LIN {X 0,Y 234.261,Z 267.411,A -85,B 0,C 180,E1 -19867.278,E2 -19867.278} C_VEL
LIN {X 0,Y 232.34,Z 276.851,A -85,B 0,C 180,E1 -19869.181,E2 -19869.181} C_VEL
LIN {X 0,Y 230.576,Z 285.695,A -85,B 0,C 180,E1 -19871.384,E2 -19871.384} C_VEL
LIN {X 0,Y 228.899,Z 293.962,A -85,B 0,C 180,E1 -19873.959,E2 -19873.959} C_VEL
LIN {X 0,Y 227.464,Z 300.726,A -85,B 0,C 180,E1 -19876.601,E2 -19876.601} C_VEL
LIN {X 0,Y 226.631,Z 306.146,A -85,B 0,C 180,E1 -19879.277,E2 -19879.277} C_VEL
LIN {X 0,Y 226.113,Z 310.355,A -85,B 0,C 180,E1 -19881.96,E2 -19881.96} C_VEL
LIN {X 0,Y 225.925,Z 313.474,A -85,B 0,C 180,E1 -19884.645,E2 -19884.645} C_VEL
LIN {X 0,Y 225.892,Z 315.003,A -85,B 0,C 180,E1 -19886.433,E2 -19886.433} C_VEL
LIN {X 0,Y 225.898,Z 316.083,A -85,B 0,C 180,E1 -19888.217,E2 -19888.217} C_VEL
LIN {X 0,Y 225.948,Z 316.728,A -85,B 0,C 180,E1 -19890,E2 -19890} C_VEL
LIN {X 0,Y 225.881,Z 316.964,A -85,B 0,C 180,E1 -19891.783,E2 -19891.783} C_VEL
LIN {X 0,Y 225.778,Z 316.356,A -85,B 0,C 180,E1 -19895.057,E2 -19895.057} C_VEL
LIN {X 0,Y 225.93,Z 315.246,A -85,B 0,C 180,E1 -19897.148,E2 -19897.148} C_VEL
LIN {X 0,Y 226.587,Z 312.1,A -85,B 0,C 180,E1 -19900.726,E2 -19900.726} C_VEL
LIN {X 0,Y 227.542,Z 308.619,A -85,B 0,C 180,E1 -19903.395,E2 -19903.395} C_VEL
LIN {X 0,Y 229.085,Z 304.112,A -85,B 0,C 180,E1 -19906.028,E2 -19906.028} C_VEL
LIN {X 0,Y 231.41,Z 297.415,A -85,B 0,C 180,E1 -19909.056,E2 -19909.056} C_VEL
LIN {X 0,Y 233.842,Z 290.185,A -85,B 0,C 180,E1 -19911.603,E2 -19911.603} C_VEL
LIN {X 0,Y 236.778,Z 281.363,A -85,B 0,C 180,E1 -19914.087,E2 -19914.087} C_VEL
LIN {X 0,Y 239.631,Z 272.445,A -85,B 0,C 180,E1 -19916.1,E2 -19916.1} C_VEL
LIN {X 0,Y 240.939,Z 262.483,A -85,B 0,C 180,E1 -19918.163,E2 -19918.163} C_VEL
LIN {X 0,Y 241.294,Z 252.576,A -85,B 0,C 180,E1 -19920.006,E2 -19920.006} C_VEL
LIN {X 0,Y 240.625,Z 241.498,A -85,B 0,C 180,E1 -19921.938,E2 -19921.938} C_VEL
LIN {X 0,Y 239.232,Z 232.018,A -85,B 0,C 180,E1 -19923.532,E2 -19923.532} C_VEL
LIN {X 0,Y 235.782,Z 218.471,A -85,B 0,C 180,E1 -19925.831,E2 -19925.831} C_VEL
LIN {X 0,Y 234.537,Z 214.79,A -85,B 0,C 180,E1 -19926.496,E2 -19926.496} C_VEL
LIN {X 0,Y 233.156,Z 210.978,A -85,B 0,C 180,E1 -19927.17,E2 -19927.17} C_VEL
LIN {X 0,Y 231.728,Z 207.641,A -85,B 0,C 180,E1 -19927.812,E2 -19927.812} C_VEL
LIN {X 0,Y 231.483,Z 206.301,A -85,B 0,C 180,E1 -19928.038,E2 -19928.038} C_VEL
LIN {X 0,Y 231.379,Z 203.886,A -85,B 0,C 180,E1 -19930.591,E2 -19930.591} C_VEL
LIN {X 0,Y 230.811,Z 200.597,A -85,B 0,C 180,E1 -19934.454,E2 -19934.454} C_VEL
LIN {X 0,Y 230.336,Z 198.024,A -85,B 0,C 180,E1 -19937.834,E2 -19937.834} C_VEL
LIN {X 0,Y 230.103,Z 196.43,A -85,B 0,C 180,E1 -19940.103,E2 -19940.103} C_VEL
LIN {X 0,Y 229.632,Z 193.775,A -85,B 0,C 180,E1 -19944.443,E2 -19944.443} C_VEL
LIN {X 0,Y 229.255,Z 191.689,A -85,B 0,C 180,E1 -19948.59,E2 -19948.59} C_VEL
LIN {X 0,Y 229.015,Z 189.98,A -85,B 0,C 180,E1 -19952.868,E2 -19952.868} C_VEL
LIN {X 0,Y 228.806,Z 188.731,A -85,B 0,C 180,E1 -19957.145,E2 -19957.145} C_VEL
LIN {X 0,Y 228.703,Z 187.823,A -85,B 0,C 180,E1 -19962.294,E2 -19962.294} C_VEL
LIN {X 0,Y 228.699,Z 187.554,A -85,B 0,C 180,E1 -19965.767,E2 -19965.767} C_VEL
LIN {X 0,Y 228.837,Z 187.534,A -85,B 0,C 180,E1 -19969.38,E2 -19969.38} C_VEL
LIN {X 0,Y 228.961,Z 187.798,A -85,B 0,C 180,E1 -19972.946,E2 -19972.946} C_VEL
LIN {X 0,Y 229.333,Z 188.636,A -85,B 0,C 180,E1 -19978.243,E2 -19978.243} C_VEL
LIN {X 0,Y 229.495,Z 189.026,A -85,B 0,C 180,E1 -19979.999,E2 -19979.999} C_VEL
LIN {X 0,Y 229.331,Z 190.067,A -85,B 0,C 180,E1 -19983.513,E2 -19983.513} C_VEL
LIN {X 0,Y 229.34,Z 191.116,A -85,B 0,C 180,E1 -19986.598,E2 -19986.598} C_VEL
LIN {X 0,Y 230.655,Z 194.258,A -85,B 0,C 180,E1 -19987.275,E2 -19987.275} C_VEL
LIN {X 0,Y 232.372,Z 196.596,A -85,B 0,C 180,E1 -19987.985,E2 -19987.985} C_VEL
LIN {X 0,Y 234.252,Z 199.958,A -85,B 0,C 180,E1 -19988.842,E2 -19988.842} C_VEL
LIN {X 0,Y 238.567,Z 209.506,A -85,B 0,C 180,E1 -19991.039,E2 -19991.039} C_VEL
LIN {X 0,Y 241.815,Z 218.493,A -85,B 0,C 180,E1 -19993.016,E2 -19993.016} C_VEL
LIN {X 0,Y 244.147,Z 227.757,A -85,B 0,C 180,E1 -19995.014,E2 -19995.014} C_VEL
LIN {X 0,Y 245.461,Z 237.244,A -85,B 0,C 180,E1 -19997.065,E2 -19997.065} C_VEL
LIN {X 0,Y 245.251,Z 239.564,A -85,B 0,C 180,E1 -19997.51,E2 -19997.51} C_VEL
LIN {X 0,Y 242.506,Z 249.033,A -85,B 0,C 180,E1 -19999.247,E2 -19999.247} C_VEL
LIN {X 0,Y 239.388,Z 258.851,A -85,B 0,C 180,E1 -20001.545,E2 -20001.545} C_VEL
LIN {X 0,Y 236.513,Z 266.907,A -85,B 0,C 180,E1 -20003.899,E2 -20003.899} C_VEL
LIN {X 0,Y 234.073,Z 273.398,A -85,B 0,C 180,E1 -20006.289,E2 -20006.289} C_VEL
LIN {X 0,Y 231.665,Z 279.237,A -85,B 0,C 180,E1 -20009.037,E2 -20009.037} C_VEL
LIN {X 0,Y 230.067,Z 282.963,A -85,B 0,C 180,E1 -20011.285,E2 -20011.285} C_VEL
LIN {X 0,Y 228.599,Z 286.233,A -85,B 0,C 180,E1 -20013.892,E2 -20013.892} C_VEL
LIN {X 0,Y 227.452,Z 288.559,A -85,B 0,C 180,E1 -20016.546,E2 -20016.546} C_VEL
LIN {X 0,Y 226.601,Z 289.931,A -85,B 0,C 180,E1 -20019.16,E2 -20019.16} C_VEL
LIN {X 0,Y 226.076,Z 290.434,A -85,B 0,C 180,E1 -20021.747,E2 -20021.747} C_VEL
LIN {X 0,Y 225.813,Z 290.119,A -85,B 0,C 180,E1 -20024.288,E2 -20024.288} C_VEL
LIN {X 0,Y 225.802,Z 289.027,A -85,B 0,C 180,E1 -20026.784,E2 -20026.784} C_VEL
LIN {X 0,Y 226.011,Z 287.146,A -85,B 0,C 180,E1 -20029.23,E2 -20029.23} C_VEL
LIN {X 0,Y 226.502,Z 284.502,A -85,B 0,C 180,E1 -20031.642,E2 -20031.642} C_VEL
LIN {X 0,Y 227.12,Z 281.132,A -85,B 0,C 180,E1 -20033.989,E2 -20033.989} C_VEL
LIN {X 0,Y 228.162,Z 275.652,A -85,B 0,C 180,E1 -20036.911,E2 -20036.911} C_VEL
LIN {X 0,Y 229.37,Z 269.303,A -85,B 0,C 180,E1 -20039.562,E2 -20039.562} C_VEL
LIN {X 0,Y 230.885,Z 262.103,A -85,B 0,C 180,E1 -20041.973,E2 -20041.973} C_VEL
LIN {X 0,Y 232.717,Z 252.954,A -85,B 0,C 180,E1 -20044.431,E2 -20044.431} C_VEL
LIN {X 0,Y 234.58,Z 242.855,A -85,B 0,C 180,E1 -20046.611,E2 -20046.611} C_VEL
LIN {X 0,Y 236.408,Z 232.431,A -85,B 0,C 180,E1 -20048.414,E2 -20048.414} C_VEL
LIN {X 0,Y 237.204,Z 227.255,A -85,B 0,C 180,E1 -20049.173,E2 -20049.173} C_VEL
LIN {X 0,Y 235.754,Z 217.735,A -85,B 0,C 180,E1 -20050.631,E2 -20050.631} C_VEL
LIN {X 0,Y 233.026,Z 205.757,A -85,B 0,C 180,E1 -20052.232,E2 -20052.232} C_VEL
LIN {X 0,Y 229.467,Z 193.019,A -85,B 0,C 180,E1 -20053.655,E2 -20053.655} C_VEL
LIN {X 0,Y 227.315,Z 185.716,A -85,B 0,C 180,E1 -20054.361,E2 -20054.361} C_VEL
LIN {X 0,Y 227.348,Z 184.804,A -85,B 0,C 180,E1 -20055.682,E2 -20055.682} C_VEL
LIN {X 0,Y 227.548,Z 184.141,A -85,B 0,C 180,E1 -20057.514,E2 -20057.514} C_VEL
LIN {X 0,Y 228.127,Z 184.067,A -85,B 0,C 180,E1 -20061.139,E2 -20061.139} C_VEL
LIN {X 0,Y 228.274,Z 184.051,A -85,B 0,C 180,E1 -20062.926,E2 -20062.926} C_VEL
LIN {X 0,Y 228.552,Z 184.018,A -85,B 0,C 180,E1 -20068.238,E2 -20068.238} C_VEL
LIN {X 0,Y 228.552,Z 184.014,A -85,B 0,C 180,E1 -20071.762,E2 -20071.762} C_VEL
LIN {X 0,Y 228.355,Z 184.04,A -85,B 0,C 180,E1 -20077.071,E2 -20077.071} C_VEL
LIN {X 0,Y 228.169,Z 184.059,A -85,B 0,C 180,E1 -20080.65,E2 -20080.65} C_VEL
LIN {X 0,Y 228.055,Z 184.078,A -85,B 0,C 180,E1 -20086.102,E2 -20086.102} C_VEL
LIN {X 0,Y 227.951,Z 184.094,A -85,B 0,C 180,E1 -20089.824,E2 -20089.824} C_VEL
LIN {X 0,Y 227.921,Z 184.096,A -85,B 0,C 180,E1 -20093.632,E2 -20093.632} C_VEL
LIN {X 0,Y 227.876,Z 184.097,A -85,B 0,C 180,E1 -20097.556,E2 -20097.556} C_VEL
LIN {X 0,Y 227.863,Z 184.102,A -85,B 0,C 180,E1 -20101.623,E2 -20101.623} C_VEL
LIN {X 0,Y 227.877,Z 184.091,A -85,B 0,C 180,E1 -20105.872,E2 -20105.872} C_VEL
LIN {X 0,Y 227.824,Z 184.104,A -85,B 0,C 180,E1 -20110.377,E2 -20110.377} C_VEL
LIN {X 0,Y 227.833,Z 184.102,A -85,B 0,C 180,E1 -20115.193,E2 -20115.193} C_VEL
LIN {X 0,Y 227.824,Z 184.099,A -85,B 0,C 180,E1 -20119.624,E2 -20119.624} C_VEL
LIN {X 0,Y 227.878,Z 184.098,A -85,B 0,C 180,E1 -20124.129,E2 -20124.129} C_VEL
LIN {X 0,Y 227.865,Z 184.098,A -85,B 0,C 180,E1 -20128.378,E2 -20128.378} C_VEL
LIN {X 0,Y 227.878,Z 184.09,A -85,B 0,C 180,E1 -20132.445,E2 -20132.445} C_VEL
LIN {X 0,Y 227.924,Z 184.093,A -85,B 0,C 180,E1 -20136.37,E2 -20136.37} C_VEL
LIN {X 0,Y 227.954,Z 184.089,A -85,B 0,C 180,E1 -20140.177,E2 -20140.177} C_VEL
LIN {X 0,Y 228.058,Z 184.067,A -85,B 0,C 180,E1 -20143.899,E2 -20143.899} C_VEL
LIN {X 0,Y 228.073,Z 184.069,A -85,B 0,C 180,E1 -20147.544,E2 -20147.544} C_VEL
LIN {X 0,Y 228.268,Z 184.049,A -85,B 0,C 180,E1 -20151.145,E2 -20151.145} C_VEL
LIN {X 0,Y 228.325,Z 184.041,A -85,B 0,C 180,E1 -20152.929,E2 -20152.929} C_VEL
LIN {X 0,Y 228.556,Z 184.007,A -85,B 0,C 180,E1 -20158.239,E2 -20158.239} C_VEL
LIN {X 0,Y 228.554,Z 184.014,A -85,B 0,C 180,E1 -20161.763,E2 -20161.763} C_VEL
LIN {X 0,Y 228.312,Z 184.04,A -85,B 0,C 180,E1 -20167.074,E2 -20167.074} C_VEL
LIN {X 0,Y 228.147,Z 184.062,A -85,B 0,C 180,E1 -20170.652,E2 -20170.652} C_VEL
LIN {X 0,Y 228.066,Z 184.075,A -85,B 0,C 180,E1 -20174.273,E2 -20174.273} C_VEL
LIN {X 0,Y 228.009,Z 184.079,A -85,B 0,C 180,E1 -20177.954,E2 -20177.954} C_VEL
LIN {X 0,Y 227.962,Z 184.087,A -85,B 0,C 180,E1 -20182.349,E2 -20182.349} C_VEL
LIN {X 0,Y 227.944,Z 184.091,A -85,B 0,C 180,E1 -20186.603,E2 -20186.603} C_VEL
LIN {X 0,Y 227.899,Z 184.096,A -85,B 0,C 180,E1 -20190.292,E2 -20190.292} C_VEL
LIN {X 0,Y 227.924,Z 184.095,A -85,B 0,C 180,E1 -20195.593,E2 -20195.593} C_VEL
LIN {X 0,Y 228.305,Z 186.122,A -85,B 0,C 180,E1 -20198.002,E2 -20198.002} C_VEL
LIN {X 0,Y 229.05,Z 190.541,A -85,B 0,C 180,E1 -20202.575,E2 -20202.575} C_VEL
LIN {X 0,Y 229.95,Z 195.263,A -85,B 0,C 180,E1 -20207.183,E2 -20207.183} C_VEL
LIN {X 0,Y 230.531,Z 198.513,A -85,B 0,C 180,E1 -20210.193,E2 -20210.193} C_VEL
LIN {X 0,Y 230.681,Z 201.082,A -85,B 0,C 180,E1 -20212.459,E2 -20212.459} C_VEL
LIN {X 0,Y 230.036,Z 204.782,A -85,B 0,C 180,E1 -20215.579,E2 -20215.579} C_VEL
LIN {X 0,Y 228.719,Z 210.452,A -85,B 0,C 180,E1 -20220.196,E2 -20220.196} C_VEL
LIN {X 0,Y 235.294,Z 214.381,A -85,B 0,C 180,E1 -20221.089,E2 -20221.089} C_VEL
LIN {X 0,Y 236.925,Z 216.569,A -85,B 0,C 180,E1 -20221.397,E2 -20221.397} C_VEL
LIN {X 0,Y 237.155,Z 218.575,A -85,B 0,C 180,E1 -20221.524,E2 -20221.524} C_VEL
LIN {X 0,Y 236.001,Z 220.936,A -85,B 0,C 180,E1 -20221.537,E2 -20221.537} C_VEL
LIN {X 0,Y 229.339,Z 226.777,A -85,B 0,C 180,E1 -20221.396,E2 -20221.396} C_VEL
LIN {X 0,Y 228.283,Z 229.366,A -85,B 0,C 180,E1 -20221.512,E2 -20221.512} C_VEL
LIN {X 0,Y 227.469,Z 232.667,A -85,B 0,C 180,E1 -20221.765,E2 -20221.765} C_VEL
LIN {X 0,Y 226.962,Z 233.889,A -85,B 0,C 180,E1 -20221.839,E2 -20221.839} C_VEL
LIN {X 0,Y 226.349,Z 238.113,A -85,B 0,C 180,E1 -20222.19,E2 -20222.19} C_VEL
LIN {X 0,Y 226.271,Z 240.519,A -85,B 0,C 180,E1 -20222.515,E2 -20222.515} C_VEL
LIN {X 0,Y 227.239,Z 253.27,A -85,B 0,C 180,E1 -20224.343,E2 -20224.343} C_VEL
LIN {X 0,Y 227.591,Z 264.718,A -85,B 0,C 180,E1 -20226.332,E2 -20226.332} C_VEL
LIN {X 0,Y 226.773,Z 270.467,A -85,B 0,C 180,E1 -20227.448,E2 -20227.448} C_VEL
LIN {X 0,Y 224.53,Z 281.068,A -85,B 0,C 180,E1 -20229.861,E2 -20229.861} C_VEL
LIN {X 0,Y 222.907,Z 288.934,A -85,B 0,C 180,E1 -20232.097,E2 -20232.097} C_VEL
LIN {X 0,Y 221.263,Z 296.609,A -85,B 0,C 180,E1 -20234.809,E2 -20234.809} C_VEL
LIN {X 0,Y 220.17,Z 301.854,A -85,B 0,C 180,E1 -20237.089,E2 -20237.089} C_VEL
LIN {X 0,Y 219.397,Z 306.936,A -85,B 0,C 180,E1 -20239.853,E2 -20239.853} C_VEL
LIN {X 0,Y 218.946,Z 310.85,A -85,B 0,C 180,E1 -20242.623,E2 -20242.623} C_VEL
LIN {X 0,Y 218.889,Z 312.852,A -85,B 0,C 180,E1 -20244.473,E2 -20244.473} C_VEL
LIN {X 0,Y 218.814,Z 314.416,A -85,B 0,C 180,E1 -20246.317,E2 -20246.317} C_VEL
LIN {X 0,Y 218.831,Z 315.561,A -85,B 0,C 180,E1 -20248.16,E2 -20248.16} C_VEL
LIN {X 0,Y 218.876,Z 316.246,A -85,B 0,C 180,E1 -20250,E2 -20250} C_VEL
LIN {X 0,Y 218.81,Z 316.516,A -85,B 0,C 180,E1 -20251.841,E2 -20251.841} C_VEL
LIN {X 0,Y 218.706,Z 316.048,A -85,B 0,C 180,E1 -20255.009,E2 -20255.009} C_VEL
LIN {X 0,Y 218.855,Z 314.95,A -85,B 0,C 180,E1 -20257.38,E2 -20257.38} C_VEL
LIN {X 0,Y 219.596,Z 311.884,A -85,B 0,C 180,E1 -20261.071,E2 -20261.071} C_VEL
LIN {X 0,Y 220.604,Z 308.487,A -85,B 0,C 180,E1 -20263.824,E2 -20263.824} C_VEL
LIN {X 0,Y 222.253,Z 304.069,A -85,B 0,C 180,E1 -20266.535,E2 -20266.535} C_VEL
LIN {X 0,Y 224.718,Z 297.526,A -85,B 0,C 180,E1 -20269.646,E2 -20269.646} C_VEL
LIN {X 0,Y 227.247,Z 290.489,A -85,B 0,C 180,E1 -20272.263,E2 -20272.263} C_VEL
LIN {X 0,Y 230.34,Z 281.824,A -85,B 0,C 180,E1 -20274.805,E2 -20274.805} C_VEL
LIN {X 0,Y 232.802,Z 274.975,A -85,B 0,C 180,E1 -20276.442,E2 -20276.442} C_VEL
LIN {X 0,Y 234.507,Z 264.948,A -85,B 0,C 180,E1 -20278.654,E2 -20278.654} C_VEL
LIN {X 0,Y 235.176,Z 255.605,A -85,B 0,C 180,E1 -20280.533,E2 -20280.533} C_VEL
LIN {X 0,Y 234.862,Z 244.628,A -85,B 0,C 180,E1 -20282.591,E2 -20282.591} C_VEL
LIN {X 0,Y 233.427,Z 233.542,A -85,B 0,C 180,E1 -20284.597,E2 -20284.597} C_VEL
LIN {X 0,Y 230.901,Z 222.438,A -85,B 0,C 180,E1 -20286.634,E2 -20286.634} C_VEL
LIN {X 0,Y 228.581,Z 215.269,A -85,B 0,C 180,E1 -20288.024,E2 -20288.024} C_VEL
LIN {X 0,Y 226.896,Z 210.971,A -85,B 0,C 180,E1 -20288.926,E2 -20288.926} C_VEL
LIN {X 0,Y 224.978,Z 207.538,A -85,B 0,C 180,E1 -20289.821,E2 -20289.821} C_VEL
LIN {X 0,Y 224.438,Z 205.627,A -85,B 0,C 180,E1 -20290.16,E2 -20290.16} C_VEL
LIN {X 0,Y 223.961,Z 202.567,A -85,B 0,C 180,E1 -20293.8,E2 -20293.8} C_VEL
LIN {X 0,Y 223.31,Z 199.009,A -85,B 0,C 180,E1 -20298.629,E2 -20298.629} C_VEL
LIN {X 0,Y 222.845,Z 196.133,A -85,B 0,C 180,E1 -20303.185,E2 -20303.185} C_VEL
LIN {X 0,Y 222.432,Z 193.89,A -85,B 0,C 180,E1 -20307.51,E2 -20307.51} C_VEL
LIN {X 0,Y 222.161,Z 192.145,A -85,B 0,C 180,E1 -20311.671,E2 -20311.671} C_VEL
LIN {X 0,Y 221.97,Z 190.858,A -85,B 0,C 180,E1 -20315.693,E2 -20315.693} C_VEL
LIN {X 0,Y 221.798,Z 189.991,A -85,B 0,C 180,E1 -20319.6,E2 -20319.6} C_VEL
LIN {X 0,Y 221.797,Z 189.451,A -85,B 0,C 180,E1 -20323.429,E2 -20323.429} C_VEL
LIN {X 0,Y 221.812,Z 189.245,A -85,B 0,C 180,E1 -20327.185,E2 -20327.185} C_VEL
LIN {X 0,Y 222.041,Z 189.293,A -85,B 0,C 180,E1 -20330.893,E2 -20330.893} C_VEL
LIN {X 0,Y 222.058,Z 189.681,A -85,B 0,C 180,E1 -20334.551,E2 -20334.551} C_VEL
LIN {X 0,Y 222.403,Z 190.237,A -85,B 0,C 180,E1 -20338.188,E2 -20338.188} C_VEL
LIN {X 0,Y 222.583,Z 190.602,A -85,B 0,C 180,E1 -20339.999,E2 -20339.999} C_VEL
LIN {X 0,Y 222.392,Z 192.036,A -85,B 0,C 180,E1 -20344.417,E2 -20344.417} C_VEL
LIN {X 0,Y 223.526,Z 194.722,A -85,B 0,C 180,E1 -20345.072,E2 -20345.072} C_VEL
LIN {X 0,Y 225.669,Z 197.315,A -85,B 0,C 180,E1 -20346.038,E2 -20346.038} C_VEL
LIN {X 0,Y 227.556,Z 200.703,A -85,B 0,C 180,E1 -20346.995,E2 -20346.995} C_VEL
LIN {X 0,Y 231.478,Z 208.431,A -85,B 0,C 180,E1 -20349.075,E2 -20349.075} C_VEL
LIN {X 0,Y 234.901,Z 217.241,A -85,B 0,C 180,E1 -20351.213,E2 -20351.213} C_VEL
LIN {X 0,Y 237.805,Z 227.826,A -85,B 0,C 180,E1 -20353.675,E2 -20353.675} C_VEL
LIN {X 0,Y 239.148,Z 236.945,A -85,B 0,C 180,E1 -20355.773,E2 -20355.773} C_VEL
LIN {X 0,Y 239.29,Z 240.746,A -85,B 0,C 180,E1 -20356.639,E2 -20356.639} C_VEL
LIN {X 0,Y 236.159,Z 250.874,A -85,B 0,C 180,E1 -20358.586,E2 -20358.586} C_VEL
LIN {X 0,Y 233.083,Z 260.012,A -85,B 0,C 180,E1 -20360.815,E2 -20360.815} C_VEL
LIN {X 0,Y 229.82,Z 268.551,A -85,B 0,C 180,E1 -20363.448,E2 -20363.448} C_VEL
LIN {X 0,Y 227.036,Z 275.302,A -85,B 0,C 180,E1 -20366.14,E2 -20366.14} C_VEL
LIN {X 0,Y 224.671,Z 280.619,A -85,B 0,C 180,E1 -20368.85,E2 -20368.85} C_VEL
LIN {X 0,Y 222.753,Z 284.694,A -85,B 0,C 180,E1 -20371.584,E2 -20371.584} C_VEL
LIN {X 0,Y 221.004,Z 288.189,A -85,B 0,C 180,E1 -20374.917,E2 -20374.917} C_VEL
LIN {X 0,Y 220.037,Z 289.79,A -85,B 0,C 180,E1 -20377.362,E2 -20377.362} C_VEL
LIN {X 0,Y 219.348,Z 290.689,A -85,B 0,C 180,E1 -20379.851,E2 -20379.851} C_VEL
LIN {X 0,Y 218.911,Z 290.874,A -85,B 0,C 180,E1 -20382.404,E2 -20382.404} C_VEL
LIN {X 0,Y 218.687,Z 290.257,A -85,B 0,C 180,E1 -20385.006,E2 -20385.006} C_VEL
LIN {X 0,Y 218.882,Z 287.826,A -85,B 0,C 180,E1 -20388.87,E2 -20388.87} C_VEL
LIN {X 0,Y 219.373,Z 285.173,A -85,B 0,C 180,E1 -20391.451,E2 -20391.451} C_VEL
LIN {X 0,Y 220.019,Z 281.636,A -85,B 0,C 180,E1 -20394.02,E2 -20394.02} C_VEL
LIN {X 0,Y 221.201,Z 275.619,A -85,B 0,C 180,E1 -20397.307,E2 -20397.307} C_VEL
LIN {X 0,Y 222.577,Z 268.83,A -85,B 0,C 180,E1 -20400.165,E2 -20400.165} C_VEL
LIN {X 0,Y 224.442,Z 260.209,A -85,B 0,C 180,E1 -20402.996,E2 -20402.996} C_VEL
LIN {X 0,Y 226.373,Z 250.803,A -85,B 0,C 180,E1 -20405.465,E2 -20405.465} C_VEL
LIN {X 0,Y 228.318,Z 240.24,A -85,B 0,C 180,E1 -20407.666,E2 -20407.666} C_VEL
LIN {X 0,Y 230.15,Z 229.581,A -85,B 0,C 180,E1 -20409.441,E2 -20409.441} C_VEL
LIN {X 0,Y 230.416,Z 227.857,A -85,B 0,C 180,E1 -20409.699,E2 -20409.699} C_VEL
LIN {X 0,Y 228.552,Z 217.131,A -85,B 0,C 180,E1 -20411.395,E2 -20411.395} C_VEL
LIN {X 0,Y 225.644,Z 204.521,A -85,B 0,C 180,E1 -20413.103,E2 -20413.103} C_VEL
LIN {X 0,Y 221.978,Z 191.691,A -85,B 0,C 180,E1 -20414.564,E2 -20414.564} C_VEL
LIN {X 0,Y 220.309,Z 186.105,A -85,B 0,C 180,E1 -20415.155,E2 -20415.155} C_VEL
LIN {X 0,Y 220.415,Z 185.029,A -85,B 0,C 180,E1 -20417.103,E2 -20417.103} C_VEL
LIN {X 0,Y 221.042,Z 184.95,A -85,B 0,C 180,E1 -20420.852,E2 -20420.852} C_VEL
LIN {X 0,Y 221.198,Z 184.933,A -85,B 0,C 180,E1 -20422.698,E2 -20422.698} C_VEL
LIN {X 0,Y 221.509,Z 184.895,A -85,B 0,C 180,E1 -20428.182,E2 -20428.182} C_VEL
LIN {X 0,Y 221.51,Z 184.892,A -85,B 0,C 180,E1 -20431.818,E2 -20431.818} C_VEL
LIN {X 0,Y 221.308,Z 184.919,A -85,B 0,C 180,E1 -20437.298,E2 -20437.298} C_VEL
LIN {X 0,Y 221.114,Z 184.938,A -85,B 0,C 180,E1 -20440.994,E2 -20440.994} C_VEL
LIN {X 0,Y 221.014,Z 184.954,A -85,B 0,C 180,E1 -20446.63,E2 -20446.63} C_VEL
LIN {X 0,Y 220.906,Z 184.969,A -85,B 0,C 180,E1 -20450.484,E2 -20450.484} C_VEL
LIN {X 0,Y 220.87,Z 184.971,A -85,B 0,C 180,E1 -20454.434,E2 -20454.434} C_VEL
LIN {X 0,Y 220.824,Z 184.975,A -85,B 0,C 180,E1 -20458.515,E2 -20458.515} C_VEL
LIN {X 0,Y 220.813,Z 184.979,A -85,B 0,C 180,E1 -20462.756,E2 -20462.756} C_VEL
LIN {X 0,Y 220.807,Z 184.973,A -85,B 0,C 180,E1 -20467.278,E2 -20467.278} C_VEL
LIN {X 0,Y 220.768,Z 184.984,A -85,B 0,C 180,E1 -20471.953,E2 -20471.953} C_VEL
LIN {X 0,Y 220.773,Z 184.979,A -85,B 0,C 180,E1 -20475.547,E2 -20475.547} C_VEL
LIN {X 0,Y 220.804,Z 184.974,A -85,B 0,C 180,E1 -20480.464,E2 -20480.464} C_VEL
LIN {X 0,Y 220.799,Z 184.981,A -85,B 0,C 180,E1 -20485.046,E2 -20485.046} C_VEL
LIN {X 0,Y 220.832,Z 184.968,A -85,B 0,C 180,E1 -20489.391,E2 -20489.391} C_VEL
LIN {X 0,Y 220.893,Z 184.962,A -85,B 0,C 180,E1 -20493.55,E2 -20493.55} C_VEL
LIN {X 0,Y 220.923,Z 184.963,A -85,B 0,C 180,E1 -20497.559,E2 -20497.559} C_VEL
LIN {X 0,Y 220.985,Z 184.95,A -85,B 0,C 180,E1 -20502.571,E2 -20502.571} C_VEL
LIN {X 0,Y 221.012,Z 184.949,A -85,B 0,C 180,E1 -20507.14,E2 -20507.14} C_VEL
LIN {X 0,Y 221.205,Z 184.929,A -85,B 0,C 180,E1 -20510.86,E2 -20510.86} C_VEL
LIN {X 0,Y 221.26,Z 184.922,A -85,B 0,C 180,E1 -20512.702,E2 -20512.702} C_VEL
LIN {X 0,Y 221.514,Z 184.883,A -85,B 0,C 180,E1 -20518.183,E2 -20518.183} C_VEL
LIN {X 0,Y 221.512,Z 184.892,A -85,B 0,C 180,E1 -20521.819,E2 -20521.819} C_VEL
LIN {X 0,Y 221.249,Z 184.92,A -85,B 0,C 180,E1 -20527.301,E2 -20527.301} C_VEL
LIN {X 0,Y 221.069,Z 184.943,A -85,B 0,C 180,E1 -20530.997,E2 -20530.997} C_VEL
LIN {X 0,Y 220.998,Z 184.955,A -85,B 0,C 180,E1 -20534.74,E2 -20534.74} C_VEL
LIN {X 0,Y 220.929,Z 184.959,A -85,B 0,C 180,E1 -20538.55,E2 -20538.55} C_VEL
LIN {X 0,Y 220.923,Z 184.964,A -85,B 0,C 180,E1 -20542.699,E2 -20542.699} C_VEL
LIN {X 0,Y 220.885,Z 184.971,A -85,B 0,C 180,E1 -20547.015,E2 -20547.015} C_VEL
LIN {X 0,Y 220.84,Z 184.976,A -85,B 0,C 180,E1 -20550.768,E2 -20550.768} C_VEL
LIN {X 0,Y 220.906,Z 185.152,A -85,B 0,C 180,E1 -20555.495,E2 -20555.495} C_VEL
LIN {X 0,Y 221.475,Z 188.638,A -85,B 0,C 180,E1 -20559.395,E2 -20559.395} C_VEL
LIN {X 0,Y 222.182,Z 192.366,A -85,B 0,C 180,E1 -20563.321,E2 -20563.321} C_VEL
LIN {X 0,Y 223.23,Z 197.73,A -85,B 0,C 180,E1 -20568.613,E2 -20568.613} C_VEL
LIN {X 0,Y 223.636,Z 201.144,A -85,B 0,C 180,E1 -20571.782,E2 -20571.782} C_VEL
LIN {X 0,Y 223.536,Z 202.861,A -85,B 0,C 180,E1 -20573.319,E2 -20573.319} C_VEL
LIN {X 0,Y 222.644,Z 206.547,A -85,B 0,C 180,E1 -20576.468,E2 -20576.468} C_VEL
LIN {X 0,Y 221.826,Z 210.15,A -85,B 0,C 180,E1 -20579.503,E2 -20579.503} C_VEL
LIN {X 0,Y 224.128,Z 223.591,A -85,B 0,C 180,E1 -20580.628,E2 -20580.628} C_VEL
LIN {X 0,Y 225.79,Z 236.167,A -85,B 0,C 180,E1 -20581.979,E2 -20581.979} C_VEL
LIN {X 0,Y 226.271,Z 240.519,A -85,B 0,C 180,E1 -20582.515,E2 -20582.515} C_VEL
LIN {X 0,Y 226.146,Z 245.933,A -85,B 0,C 180,E1 -20583.192,E2 -20583.192} C_VEL
LIN {X 0,Y 224.193,Z 254.653,A -85,B 0,C 180,E1 -20584.319,E2 -20584.319} C_VEL
LIN {X 0,Y 222.077,Z 261.222,A -85,B 0,C 180,E1 -20585.304,E2 -20585.304} C_VEL
LIN {X 0,Y 220.431,Z 267.55,A -85,B 0,C 180,E1 -20586.438,E2 -20586.438} C_VEL
LIN {X 0,Y 218.589,Z 276.154,A -85,B 0,C 180,E1 -20588.3,E2 -20588.3} C_VEL
LIN {X 0,Y 216.706,Z 284.693,A -85,B 0,C 180,E1 -20590.555,E2 -20590.555} C_VEL
LIN {X 0,Y 214.888,Z 293.204,A -85,B 0,C 180,E1 -20593.371,E2 -20593.371} C_VEL
LIN {X 0,Y 213.39,Z 299.949,A -85,B 0,C 180,E1 -20596.186,E2 -20596.186} C_VEL
LIN {X 0,Y 212.383,Z 306.154,A -85,B 0,C 180,E1 -20599.514,E2 -20599.514} C_VEL
LIN {X 0,Y 211.911,Z 310.155,A -85,B 0,C 180,E1 -20602.377,E2 -20602.377} C_VEL
LIN {X 0,Y 211.796,Z 312.458,A -85,B 0,C 180,E1 -20604.563,E2 -20604.563} C_VEL
LIN {X 0,Y 211.764,Z 314.996,A -85,B 0,C 180,E1 -20608.098,E2 -20608.098} C_VEL
LIN {X 0,Y 211.805,Z 315.756,A -85,B 0,C 180,E1 -20610,E2 -20610} C_VEL
LIN {X 0,Y 211.74,Z 316.065,A -85,B 0,C 180,E1 -20611.902,E2 -20611.902} C_VEL
LIN {X 0,Y 211.635,Z 315.505,A -85,B 0,C 180,E1 -20615.718,E2 -20615.718} C_VEL
LIN {X 0,Y 211.788,Z 314.646,A -85,B 0,C 180,E1 -20617.628,E2 -20617.628} C_VEL
LIN {X 0,Y 212.582,Z 311.668,A -85,B 0,C 180,E1 -20621.442,E2 -20621.442} C_VEL
LIN {X 0,Y 213.691,Z 308.375,A -85,B 0,C 180,E1 -20624.281,E2 -20624.281} C_VEL
LIN {X 0,Y 215.445,Z 304.078,A -85,B 0,C 180,E1 -20627.073,E2 -20627.073} C_VEL
LIN {X 0,Y 218.053,Z 297.651,A -85,B 0,C 180,E1 -20630.273,E2 -20630.273} C_VEL
LIN {X 0,Y 220.694,Z 290.76,A -85,B 0,C 180,E1 -20632.961,E2 -20632.961} C_VEL
LIN {X 0,Y 223.943,Z 282.284,A -85,B 0,C 180,E1 -20635.564,E2 -20635.564} C_VEL
LIN {X 0,Y 226.487,Z 275.599,A -85,B 0,C 180,E1 -20637.239,E2 -20637.239} C_VEL
LIN {X 0,Y 228.317,Z 265.958,A -85,B 0,C 180,E1 -20639.506,E2 -20639.506} C_VEL
LIN {X 0,Y 229.109,Z 256.905,A -85,B 0,C 180,E1 -20641.432,E2 -20641.432} C_VEL
LIN {X 0,Y 229.013,Z 246.387,A -85,B 0,C 180,E1 -20643.532,E2 -20643.532} C_VEL
LIN {X 0,Y 227.864,Z 235.774,A -85,B 0,C 180,E1 -20645.606,E2 -20645.606} C_VEL
LIN {X 0,Y 225.52,Z 224.268,A -85,B 0,C 180,E1 -20647.86,E2 -20647.86} C_VEL
LIN {X 0,Y 222.576,Z 215.757,A -85,B 0,C 180,E1 -20649.763,E2 -20649.763} C_VEL
LIN {X 0,Y 220.782,Z 211.983,A -85,B 0,C 180,E1 -20650.745,E2 -20650.745} C_VEL
LIN {X 0,Y 220.124,Z 210.614,A -85,B 0,C 180,E1 -20651.106,E2 -20651.106} C_VEL
LIN {X 0,Y 217.99,Z 207.341,A -85,B 0,C 180,E1 -20652.209,E2 -20652.209} C_VEL
LIN {X 0,Y 217.158,Z 204.78,A -85,B 0,C 180,E1 -20652.816,E2 -20652.816} C_VEL
LIN {X 0,Y 216.526,Z 201.653,A -85,B 0,C 180,E1 -20657.029,E2 -20657.029} C_VEL
LIN {X 0,Y 216.07,Z 198.552,A -85,B 0,C 180,E1 -20661.828,E2 -20661.828} C_VEL
LIN {X 0,Y 215.62,Z 196.134,A -85,B 0,C 180,E1 -20666.35,E2 -20666.35} C_VEL
LIN {X 0,Y 215.328,Z 194.248,A -85,B 0,C 180,E1 -20670.686,E2 -20670.686} C_VEL
LIN {X 0,Y 215.104,Z 192.851,A -85,B 0,C 180,E1 -20674.865,E2 -20674.865} C_VEL
LIN {X 0,Y 214.94,Z 191.878,A -85,B 0,C 180,E1 -20678.919,E2 -20678.919} C_VEL
LIN {X 0,Y 214.918,Z 191.261,A -85,B 0,C 180,E1 -20682.883,E2 -20682.883} C_VEL
LIN {X 0,Y 214.916,Z 190.994,A -85,B 0,C 180,E1 -20686.766,E2 -20686.766} C_VEL
LIN {X 0,Y 215.128,Z 190.992,A -85,B 0,C 180,E1 -20690.598,E2 -20690.598} C_VEL
LIN {X 0,Y 215.152,Z 191.318,A -85,B 0,C 180,E1 -20694.375,E2 -20694.375} C_VEL
LIN {X 0,Y 215.487,Z 191.84,A -85,B 0,C 180,E1 -20698.13,E2 -20698.13} C_VEL
LIN {X 0,Y 215.685,Z 192.191,A -85,B 0,C 180,E1 -20699.999,E2 -20699.999} C_VEL
LIN {X 0,Y 215.587,Z 192.672,A -85,B 0,C 180,E1 -20701.867,E2 -20701.867} C_VEL
LIN {X 0,Y 216.643,Z 195.447,A -85,B 0,C 180,E1 -20702.625,E2 -20702.625} C_VEL
LIN {X 0,Y 218.931,Z 198.168,A -85,B 0,C 180,E1 -20703.795,E2 -20703.795} C_VEL
LIN {X 0,Y 220.736,Z 201.437,A -85,B 0,C 180,E1 -20704.85,E2 -20704.85} C_VEL
LIN {X 0,Y 221.888,Z 203.044,A -85,B 0,C 180,E1 -20705.452,E2 -20705.452} C_VEL
LIN {X 0,Y 225.765,Z 210.495,A -85,B 0,C 180,E1 -20707.714,E2 -20707.714} C_VEL
LIN {X 0,Y 229.732,Z 221.368,A -85,B 0,C 180,E1 -20710.576,E2 -20710.576} C_VEL
LIN {X 0,Y 232.198,Z 231.516,A -85,B 0,C 180,E1 -20713.12,E2 -20713.12} C_VEL
LIN {X 0,Y 233.248,Z 240.724,A -85,B 0,C 180,E1 -20715.377,E2 -20715.377} C_VEL
LIN {X 0,Y 233.316,Z 242.117,A -85,B 0,C 180,E1 -20715.729,E2 -20715.729} C_VEL
LIN {X 0,Y 230.026,Z 252.304,A -85,B 0,C 180,E1 -20717.789,E2 -20717.789} C_VEL
LIN {X 0,Y 226.986,Z 260.693,A -85,B 0,C 180,E1 -20719.912,E2 -20719.912} C_VEL
LIN {X 0,Y 223.692,Z 268.839,A -85,B 0,C 180,E1 -20722.473,E2 -20722.473} C_VEL
LIN {X 0,Y 220.609,Z 275.875,A -85,B 0,C 180,E1 -20725.344,E2 -20725.344} C_VEL
LIN {X 0,Y 218.331,Z 280.644,A -85,B 0,C 180,E1 -20727.822,E2 -20727.822} C_VEL
LIN {X 0,Y 215.727,Z 285.788,A -85,B 0,C 180,E1 -20731.415,E2 -20731.415} C_VEL
LIN {X 0,Y 213.946,Z 288.97,A -85,B 0,C 180,E1 -20734.79,E2 -20734.79} C_VEL
LIN {X 0,Y 212.869,Z 290.586,A -85,B 0,C 180,E1 -20737.591,E2 -20737.591} C_VEL
LIN {X 0,Y 212.162,Z 291.313,A -85,B 0,C 180,E1 -20740.368,E2 -20740.368} C_VEL
LIN {X 0,Y 211.643,Z 290.879,A -85,B 0,C 180,E1 -20744.213,E2 -20744.213} C_VEL
LIN {X 0,Y 211.601,Z 289.604,A -85,B 0,C 180,E1 -20746.943,E2 -20746.943} C_VEL
LIN {X 0,Y 211.929,Z 287.456,A -85,B 0,C 180,E1 -20749.703,E2 -20749.703} C_VEL
LIN {X 0,Y 212.528,Z 284.295,A -85,B 0,C 180,E1 -20752.526,E2 -20752.526} C_VEL
LIN {X 0,Y 213.525,Z 278.955,A -85,B 0,C 180,E1 -20755.975,E2 -20755.975} C_VEL
LIN {X 0,Y 214.823,Z 272.786,A -85,B 0,C 180,E1 -20758.999,E2 -20758.999} C_VEL
LIN {X 0,Y 216.491,Z 265.144,A -85,B 0,C 180,E1 -20761.919,E2 -20761.919} C_VEL
LIN {X 0,Y 218.279,Z 257.17,A -85,B 0,C 180,E1 -20764.357,E2 -20764.357} C_VEL
LIN {X 0,Y 220.222,Z 247.669,A -85,B 0,C 180,E1 -20766.719,E2 -20766.719} C_VEL
LIN {X 0,Y 221.988,Z 238.109,A -85,B 0,C 180,E1 -20768.648,E2 -20768.648} C_VEL
LIN {X 0,Y 223.569,Z 228.392,A -85,B 0,C 180,E1 -20770.249,E2 -20770.249} C_VEL
LIN {X 0,Y 221.667,Z 217.854,A -85,B 0,C 180,E1 -20771.993,E2 -20771.993} C_VEL
LIN {X 0,Y 218.959,Z 205.912,A -85,B 0,C 180,E1 -20773.689,E2 -20773.689} C_VEL
LIN {X 0,Y 215.219,Z 192.714,A -85,B 0,C 180,E1 -20775.28,E2 -20775.28} C_VEL
LIN {X 0,Y 213.268,Z 186.545,A -85,B 0,C 180,E1 -20775.934,E2 -20775.934} C_VEL
LIN {X 0,Y 213.317,Z 186.055,A -85,B 0,C 180,E1 -20776.666,E2 -20776.666} C_VEL
LIN {X 0,Y 213.978,Z 185.832,A -85,B 0,C 180,E1 -20780.548,E2 -20780.548} C_VEL
LIN {X 0,Y 214.124,Z 185.816,A -85,B 0,C 180,E1 -20782.456,E2 -20782.456} C_VEL
LIN {X 0,Y 214.443,Z 185.775,A -85,B 0,C 180,E1 -20788.122,E2 -20788.122} C_VEL
LIN {X 0,Y 214.552,Z 185.759,A -85,B 0,C 180,E1 -20790,E2 -20790} C_VEL
LIN {X 0,Y 214.444,Z 185.772,A -85,B 0,C 180,E1 -20791.878,E2 -20791.878} C_VEL
LIN {X 0,Y 214.245,Z 185.8,A -85,B 0,C 180,E1 -20797.539,E2 -20797.539} C_VEL
LIN {X 0,Y 214.045,Z 185.82,A -85,B 0,C 180,E1 -20801.362,E2 -20801.362} C_VEL
LIN {X 0,Y 213.931,Z 185.84,A -85,B 0,C 180,E1 -20805.237,E2 -20805.237} C_VEL
LIN {X 0,Y 213.873,Z 185.843,A -85,B 0,C 180,E1 -20809.184,E2 -20809.184} C_VEL
LIN {X 0,Y 213.853,Z 185.85,A -85,B 0,C 180,E1 -20813.226,E2 -20813.226} C_VEL
LIN {X 0,Y 213.826,Z 185.846,A -85,B 0,C 180,E1 -20817.45,E2 -20817.45} C_VEL
LIN {X 0,Y 213.764,Z 185.858,A -85,B 0,C 180,E1 -20821.738,E2 -20821.738} C_VEL
LIN {X 0,Y 213.74,Z 185.85,A -85,B 0,C 180,E1 -20826.289,E2 -20826.289} C_VEL
LIN {X 0,Y 213.71,Z 185.865,A -85,B 0,C 180,E1 -20831.126,E2 -20831.126} C_VEL
LIN {X 0,Y 213.705,Z 185.863,A -85,B 0,C 180,E1 -20833.679,E2 -20833.679} C_VEL
LIN {X 0,Y 213.705,Z 185.859,A -85,B 0,C 180,E1 -20836.344,E2 -20836.344} C_VEL
LIN {X 0,Y 213.715,Z 185.854,A -85,B 0,C 180,E1 -20839.143,E2 -20839.143} C_VEL
LIN {X 0,Y 213.741,Z 185.858,A -85,B 0,C 180,E1 -20843.712,E2 -20843.712} C_VEL
LIN {X 0,Y 213.779,Z 185.849,A -85,B 0,C 180,E1 -20848.732,E2 -20848.732} C_VEL
LIN {X 0,Y 213.825,Z 185.84,A -85,B 0,C 180,E1 -20852.604,E2 -20852.604} C_VEL
LIN {X 0,Y 213.861,Z 185.844,A -85,B 0,C 180,E1 -20856.947,E2 -20856.947} C_VEL
LIN {X 0,Y 213.933,Z 185.83,A -85,B 0,C 180,E1 -20862.305,E2 -20862.305} C_VEL
LIN {X 0,Y 213.953,Z 185.829,A -85,B 0,C 180,E1 -20866.708,E2 -20866.708} C_VEL
LIN {X 0,Y 214.142,Z 185.811,A -85,B 0,C 180,E1 -20870.556,E2 -20870.556} C_VEL
LIN {X 0,Y 214.102,Z 185.811,A -85,B 0,C 180,E1 -20874.35,E2 -20874.35} C_VEL
LIN {X 0,Y 214.447,Z 185.762,A -85,B 0,C 180,E1 -20878.123,E2 -20878.123} C_VEL
LIN {X 0,Y 214.551,Z 185.755,A -85,B 0,C 180,E1 -20880.001,E2 -20880.001} C_VEL
LIN {X 0,Y 214.445,Z 185.772,A -85,B 0,C 180,E1 -20881.879,E2 -20881.879} C_VEL
LIN {X 0,Y 214.19,Z 185.8,A -85,B 0,C 180,E1 -20887.543,E2 -20887.543} C_VEL
LIN {X 0,Y 214,Z 185.825,A -85,B 0,C 180,E1 -20891.365,E2 -20891.365} C_VEL
LIN {X 0,Y 213.936,Z 185.836,A -85,B 0,C 180,E1 -20895.238,E2 -20895.238} C_VEL
LIN {X 0,Y 213.878,Z 185.838,A -85,B 0,C 180,E1 -20899.185,E2 -20899.185} C_VEL
LIN {X 0,Y 213.858,Z 185.846,A -85,B 0,C 180,E1 -20903.227,E2 -20903.227} C_VEL
LIN {X 0,Y 213.831,Z 185.852,A -85,B 0,C 180,E1 -20907.451,E2 -20907.451} C_VEL
LIN {X 0,Y 213.769,Z 185.858,A -85,B 0,C 180,E1 -20911.738,E2 -20911.738} C_VEL
LIN {X 0,Y 213.863,Z 186.004,A -85,B 0,C 180,E1 -20914.99,E2 -20914.99} C_VEL
LIN {X 0,Y 214.543,Z 190.099,A -85,B 0,C 180,E1 -20919.702,E2 -20919.702} C_VEL
LIN {X 0,Y 215.279,Z 194.185,A -85,B 0,C 180,E1 -20924.093,E2 -20924.093} C_VEL
LIN {X 0,Y 216.151,Z 198.437,A -85,B 0,C 180,E1 -20928.404,E2 -20928.404} C_VEL
LIN {X 0,Y 216.552,Z 202.097,A -85,B 0,C 180,E1 -20931.93,E2 -20931.93} C_VEL
LIN {X 0,Y 216.162,Z 204.795,A -85,B 0,C 180,E1 -20934.373,E2 -20934.373} C_VEL
LIN {X 0,Y 214.942,Z 209.738,A -85,B 0,C 180,E1 -20938.711,E2 -20938.711} C_VEL
LIN {X 0,Y 217.053,Z 222.277,A -85,B 0,C 180,E1 -20939.798,E2 -20939.798} C_VEL
LIN {X 0,Y 218.768,Z 234.955,A -85,B 0,C 180,E1 -20941.192,E2 -20941.192} C_VEL
LIN {X 0,Y 219.874,Z 246.324,A -85,B 0,C 180,E1 -20942.724,E2 -20942.724} C_VEL
LIN {X 0,Y 220.511,Z 257.435,A -85,B 0,C 180,E1 -20944.516,E2 -20944.516} C_VEL
LIN {X 0,Y 220.572,Z 266.74,A -85,B 0,C 180,E1 -20946.28,E2 -20946.28} C_VEL
LIN {X 0,Y 220.431,Z 267.55,A -85,B 0,C 180,E1 -20946.438,E2 -20946.438} C_VEL
LIN {X 0,Y 218.954,Z 272.104,A -85,B 0,C 180,E1 -20947.334,E2 -20947.334} C_VEL
LIN {X 0,Y 214.717,Z 279.03,A -85,B 0,C 180,E1 -20948.83,E2 -20948.83} C_VEL
LIN {X 0,Y 210.358,Z 285.397,A -85,B 0,C 180,E1 -20950.523,E2 -20950.523} C_VEL
LIN {X 0,Y 208.725,Z 289.087,A -85,B 0,C 180,E1 -20951.713,E2 -20951.713} C_VEL
LIN {X 0,Y 206.961,Z 296.877,A -85,B 0,C 180,E1 -20954.742,E2 -20954.742} C_VEL
LIN {X 0,Y 205.643,Z 303.701,A -85,B 0,C 180,E1 -20958.168,E2 -20958.168} C_VEL
LIN {X 0,Y 204.981,Z 308.175,A -85,B 0,C 180,E1 -20961.125,E2 -20961.125} C_VEL
LIN {X 0,Y 204.723,Z 312.005,A -85,B 0,C 180,E1 -20964.602,E2 -20964.602} C_VEL
LIN {X 0,Y 204.698,Z 314.425,A -85,B 0,C 180,E1 -20968.033,E2 -20968.033} C_VEL
LIN {X 0,Y 204.737,Z 315.244,A -85,B 0,C 180,E1 -20970,E2 -20970} C_VEL
LIN {X 0,Y 204.669,Z 315.615,A -85,B 0,C 180,E1 -20971.968,E2 -20971.968} C_VEL
LIN {X 0,Y 204.568,Z 315.132,A -85,B 0,C 180,E1 -20975.916,E2 -20975.916} C_VEL
LIN {X 0,Y 205.061,Z 313.118,A -85,B 0,C 180,E1 -20979.868,E2 -20979.868} C_VEL
LIN {X 0,Y 206.306,Z 309.45,A -85,B 0,C 180,E1 -20983.796,E2 -20983.796} C_VEL
LIN {X 0,Y 207.97,Z 305.592,A -85,B 0,C 180,E1 -20986.693,E2 -20986.693} C_VEL
LIN {X 0,Y 210.074,Z 300.673,A -85,B 0,C 180,E1 -20989.546,E2 -20989.546} C_VEL
LIN {X 0,Y 212.967,Z 294.056,A -85,B 0,C 180,E1 -20992.545,E2 -20992.545} C_VEL
LIN {X 0,Y 215.805,Z 287.149,A -85,B 0,C 180,E1 -20995.048,E2 -20995.048} C_VEL
LIN {X 0,Y 218.938,Z 279.661,A -85,B 0,C 180,E1 -20997.222,E2 -20997.222} C_VEL
LIN {X 0,Y 220.658,Z 274.554,A -85,B 0,C 180,E1 -20998.539,E2 -20998.539} C_VEL
LIN {X 0,Y 222.552,Z 264.222,A -85,B 0,C 180,E1 -21001.015,E2 -21001.015} C_VEL
LIN {X 0,Y 223.254,Z 254.609,A -85,B 0,C 180,E1 -21003.15,E2 -21003.15} C_VEL
LIN {X 0,Y 222.954,Z 243.592,A -85,B 0,C 180,E1 -21005.469,E2 -21005.469} C_VEL
LIN {X 0,Y 221.358,Z 231.731,A -85,B 0,C 180,E1 -21007.962,E2 -21007.962} C_VEL
LIN {X 0,Y 219.394,Z 223.818,A -85,B 0,C 180,E1 -21009.752,E2 -21009.752} C_VEL
LIN {X 0,Y 216.285,Z 215.964,A -85,B 0,C 180,E1 -21011.853,E2 -21011.853} C_VEL
LIN {X 0,Y 214.148,Z 212.198,A -85,B 0,C 180,E1 -21013.129,E2 -21013.129} C_VEL
LIN {X 0,Y 213.293,Z 210.239,A -85,B 0,C 180,E1 -21013.682,E2 -21013.682} C_VEL
LIN {X 0,Y 210.752,Z 206.743,A -85,B 0,C 180,E1 -21015.177,E2 -21015.177} C_VEL
LIN {X 0,Y 209.716,Z 203.876,A -85,B 0,C 180,E1 -21016.001,E2 -21016.001} C_VEL
LIN {X 0,Y 209.243,Z 200.896,A -85,B 0,C 180,E1 -21020.581,E2 -21020.581} C_VEL
LIN {X 0,Y 208.813,Z 198.421,A -85,B 0,C 180,E1 -21025.097,E2 -21025.097} C_VEL
LIN {X 0,Y 208.493,Z 196.388,A -85,B 0,C 180,E1 -21029.626,E2 -21029.626} C_VEL
LIN {X 0,Y 208.27,Z 194.855,A -85,B 0,C 180,E1 -21033.979,E2 -21033.979} C_VEL
LIN {X 0,Y 208.232,Z 194.257,A -85,B 0,C 180,E1 -21036.107,E2 -21036.107} C_VEL
LIN {X 0,Y 208.056,Z 193.082,A -85,B 0,C 180,E1 -21042.3,E2 -21042.3} C_VEL
LIN {X 0,Y 208.034,Z 192.743,A -85,B 0,C 180,E1 -21046.32,E2 -21046.32} C_VEL
LIN {X 0,Y 208.212,Z 192.686,A -85,B 0,C 180,E1 -21050.283,E2 -21050.283} C_VEL
LIN {X 0,Y 208.263,Z 192.97,A -85,B 0,C 180,E1 -21054.189,E2 -21054.189} C_VEL
LIN {X 0,Y 208.631,Z 193.607,A -85,B 0,C 180,E1 -21058.793,E2 -21058.793} C_VEL
LIN {X 0,Y 209.789,Z 196.159,A -85,B 0,C 180,E1 -21059.699,E2 -21059.699} C_VEL
LIN {X 0,Y 212.441,Z 199.243,A -85,B 0,C 180,E1 -21061.302,E2 -21061.302} C_VEL
LIN {X 0,Y 214.307,Z 202.65,A -85,B 0,C 180,E1 -21062.583,E2 -21062.583} C_VEL
LIN {X 0,Y 215.378,Z 204.108,A -85,B 0,C 180,E1 -21063.214,E2 -21063.214} C_VEL
LIN {X 0,Y 218.865,Z 210.436,A -85,B 0,C 180,E1 -21065.465,E2 -21065.465} C_VEL
LIN {X 0,Y 222.07,Z 217.65,A -85,B 0,C 180,E1 -21067.729,E2 -21067.729} C_VEL
LIN {X 0,Y 224.72,Z 226.197,A -85,B 0,C 180,E1 -21070.131,E2 -21070.131} C_VEL
LIN {X 0,Y 226.582,Z 235.192,A -85,B 0,C 180,E1 -21072.539,E2 -21072.539} C_VEL
LIN {X 0,Y 227.25,Z 243.84,A -85,B 0,C 180,E1 -21074.827,E2 -21074.827} C_VEL
LIN {X 0,Y 226.161,Z 247.488,A -85,B 0,C 180,E1 -21075.562,E2 -21075.562} C_VEL
LIN {X 0,Y 222.721,Z 257.064,A -85,B 0,C 180,E1 -21077.759,E2 -21077.759} C_VEL
LIN {X 0,Y 219.313,Z 265.393,A -85,B 0,C 180,E1 -21080.15,E2 -21080.15} C_VEL
LIN {X 0,Y 215.805,Z 273.125,A -85,B 0,C 180,E1 -21083.003,E2 -21083.003} C_VEL
LIN {X 0,Y 212.761,Z 279.329,A -85,B 0,C 180,E1 -21085.965,E2 -21085.965} C_VEL
LIN {X 0,Y 210.537,Z 283.608,A -85,B 0,C 180,E1 -21088.624,E2 -21088.624} C_VEL
LIN {X 0,Y 208.657,Z 286.909,A -85,B 0,C 180,E1 -21091.306,E2 -21091.306} C_VEL
LIN {X 0,Y 207.857,Z 288.294,A -85,B 0,C 180,E1 -21092.75,E2 -21092.75} C_VEL
LIN {X 0,Y 206.601,Z 290.196,A -85,B 0,C 180,E1 -21095.329,E2 -21095.329} C_VEL
LIN {X 0,Y 205.601,Z 291.415,A -85,B 0,C 180,E1 -21098.167,E2 -21098.167} C_VEL
LIN {X 0,Y 204.946,Z 291.792,A -85,B 0,C 180,E1 -21101.024,E2 -21101.024} C_VEL
LIN {X 0,Y 204.588,Z 291.357,A -85,B 0,C 180,E1 -21103.83,E2 -21103.83} C_VEL
LIN {X 0,Y 204.524,Z 290.153,A -85,B 0,C 180,E1 -21106.586,E2 -21106.586} C_VEL
LIN {X 0,Y 204.773,Z 288.185,A -85,B 0,C 180,E1 -21109.299,E2 -21109.299} C_VEL
LIN {X 0,Y 205.29,Z 285.424,A -85,B 0,C 180,E1 -21111.959,E2 -21111.959} C_VEL
LIN {X 0,Y 206.064,Z 281.334,A -85,B 0,C 180,E1 -21114.937,E2 -21114.937} C_VEL
LIN {X 0,Y 207.217,Z 275.898,A -85,B 0,C 180,E1 -21117.982,E2 -21117.982} C_VEL
LIN {X 0,Y 208.773,Z 268.793,A -85,B 0,C 180,E1 -21121.072,E2 -21121.072} C_VEL
LIN {X 0,Y 210.856,Z 259.771,A -85,B 0,C 180,E1 -21124.147,E2 -21124.147} C_VEL
LIN {X 0,Y 212.887,Z 250.418,A -85,B 0,C 180,E1 -21126.662,E2 -21126.662} C_VEL
LIN {X 0,Y 214.935,Z 239.954,A -85,B 0,C 180,E1 -21128.919,E2 -21128.919} C_VEL
LIN {X 0,Y 216.735,Z 230.057,A -85,B 0,C 180,E1 -21130.636,E2 -21130.636} C_VEL
LIN {X 0,Y 215.339,Z 221.261,A -85,B 0,C 180,E1 -21132.183,E2 -21132.183} C_VEL
LIN {X 0,Y 212.875,Z 209.843,A -85,B 0,C 180,E1 -21133.948,E2 -21133.948} C_VEL
LIN {X 0,Y 209.606,Z 197.585,A -85,B 0,C 180,E1 -21135.558,E2 -21135.558} C_VEL
LIN {X 0,Y 206.286,Z 186.961,A -85,B 0,C 180,E1 -21136.767,E2 -21136.767} C_VEL
LIN {X 0,Y 206.855,Z 186.721,A -85,B 0,C 180,E1 -21140.219,E2 -21140.219} C_VEL
LIN {X 0,Y 207.056,Z 186.696,A -85,B 0,C 180,E1 -21142.196,E2 -21142.196} C_VEL
LIN {X 0,Y 207.379,Z 186.654,A -85,B 0,C 180,E1 -21148.058,E2 -21148.058} C_VEL
LIN {X 0,Y 207.516,Z 186.635,A -85,B 0,C 180,E1 -21150,E2 -21150} C_VEL
LIN {X 0,Y 207.085,Z 186.689,A -85,B 0,C 180,E1 -21153.892,E2 -21153.892} C_VEL
LIN {X 0,Y 207.186,Z 186.681,A -85,B 0,C 180,E1 -21157.798,E2 -21157.798} C_VEL
LIN {X 0,Y 206.98,Z 186.703,A -85,B 0,C 180,E1 -21161.755,E2 -21161.755} C_VEL
LIN {X 0,Y 206.865,Z 186.72,A -85,B 0,C 180,E1 -21165.771,E2 -21165.771} C_VEL
LIN {X 0,Y 206.81,Z 186.727,A -85,B 0,C 180,E1 -21169.866,E2 -21169.866} C_VEL
LIN {X 0,Y 206.765,Z 186.729,A -85,B 0,C 180,E1 -21174.072,E2 -21174.072} C_VEL
LIN {X 0,Y 206.734,Z 186.73,A -85,B 0,C 180,E1 -21178.42,E2 -21178.42} C_VEL
LIN {X 0,Y 206.695,Z 186.739,A -85,B 0,C 180,E1 -21182.958,E2 -21182.958} C_VEL
LIN {X 0,Y 206.677,Z 186.734,A -85,B 0,C 180,E1 -21187.74,E2 -21187.74} C_VEL
LIN {X 0,Y 206.64,Z 186.745,A -85,B 0,C 180,E1 -21191.564,E2 -21191.564} C_VEL
LIN {X 0,Y 206.632,Z 186.74,A -85,B 0,C 180,E1 -21195.582,E2 -21195.582} C_VEL
LIN {X 0,Y 206.658,Z 186.734,A -85,B 0,C 180,E1 -21199.75,E2 -21199.75} C_VEL
LIN {X 0,Y 206.697,Z 186.739,A -85,B 0,C 180,E1 -21204.69,E2 -21204.69} C_VEL
LIN {X 0,Y 206.705,Z 186.726,A -85,B 0,C 180,E1 -21209.337,E2 -21209.337} C_VEL
LIN {X 0,Y 206.733,Z 186.725,A -85,B 0,C 180,E1 -21213.773,E2 -21213.773} C_VEL
LIN {X 0,Y 206.777,Z 186.727,A -85,B 0,C 180,E1 -21218.047,E2 -21218.047} C_VEL
LIN {X 0,Y 206.878,Z 186.709,A -85,B 0,C 180,E1 -21222.198,E2 -21222.198} C_VEL
LIN {X 0,Y 206.896,Z 186.703,A -85,B 0,C 180,E1 -21226.245,E2 -21226.245} C_VEL
LIN {X 0,Y 207.099,Z 186.688,A -85,B 0,C 180,E1 -21230.232,E2 -21230.232} C_VEL
LIN {X 0,Y 207.063,Z 186.689,A -85,B 0,C 180,E1 -21234.157,E2 -21234.157} C_VEL
LIN {X 0,Y 207.383,Z 186.641,A -85,B 0,C 180,E1 -21238.059,E2 -21238.059} C_VEL
LIN {X 0,Y 207.516,Z 186.631,A -85,B 0,C 180,E1 -21240.001,E2 -21240.001} C_VEL
LIN {X 0,Y 207.381,Z 186.652,A -85,B 0,C 180,E1 -21241.943,E2 -21241.943} C_VEL
LIN {X 0,Y 207.133,Z 186.676,A -85,B 0,C 180,E1 -21247.801,E2 -21247.801} C_VEL
LIN {X 0,Y 206.926,Z 186.708,A -85,B 0,C 180,E1 -21251.759,E2 -21251.759} C_VEL
LIN {X 0,Y 206.869,Z 186.715,A -85,B 0,C 180,E1 -21255.772,E2 -21255.772} C_VEL
LIN {X 0,Y 206.815,Z 186.722,A -85,B 0,C 180,E1 -21259.867,E2 -21259.867} C_VEL
LIN {X 0,Y 206.77,Z 186.728,A -85,B 0,C 180,E1 -21264.072,E2 -21264.072} C_VEL
LIN {X 0,Y 206.739,Z 186.733,A -85,B 0,C 180,E1 -21268.421,E2 -21268.421} C_VEL
LIN {X 0,Y 206.712,Z 186.737,A -85,B 0,C 180,E1 -21272.956,E2 -21272.956} C_VEL
LIN {X 0,Y 206.787,Z 186.803,A -85,B 0,C 180,E1 -21274.405,E2 -21274.405} C_VEL
LIN {X 0,Y 207.383,Z 190.462,A -85,B 0,C 180,E1 -21278.791,E2 -21278.791} C_VEL
LIN {X 0,Y 208.205,Z 194.861,A -85,B 0,C 180,E1 -21283.698,E2 -21283.698} C_VEL
LIN {X 0,Y 208.959,Z 198.665,A -85,B 0,C 180,E1 -21287.727,E2 -21287.727} C_VEL
LIN {X 0,Y 209.5,Z 202.649,A -85,B 0,C 180,E1 -21291.713,E2 -21291.713} C_VEL
LIN {X 0,Y 209.228,Z 204.787,A -85,B 0,C 180,E1 -21293.724,E2 -21293.724} C_VEL
LIN {X 0,Y 208.049,Z 209.361,A -85,B 0,C 180,E1 -21297.888,E2 -21297.888} C_VEL
LIN {X 0,Y 210.334,Z 222.591,A -85,B 0,C 180,E1 -21299.083,E2 -21299.083} C_VEL
LIN {X 0,Y 211.998,Z 235.568,A -85,B 0,C 180,E1 -21300.594,E2 -21300.594} C_VEL
LIN {X 0,Y 213.057,Z 247.192,A -85,B 0,C 180,E1 -21302.25,E2 -21302.25} C_VEL
LIN {X 0,Y 213.634,Z 258.826,A -85,B 0,C 180,E1 -21304.236,E2 -21304.236} C_VEL
LIN {X 0,Y 213.545,Z 267.582,A -85,B 0,C 180,E1 -21305.998,E2 -21305.998} C_VEL
LIN {X 0,Y 211.552,Z 276.671,A -85,B 0,C 180,E1 -21308.054,E2 -21308.054} C_VEL
LIN {X 0,Y 209.621,Z 285.121,A -85,B 0,C 180,E1 -21310.411,E2 -21310.411} C_VEL
LIN {X 0,Y 208.725,Z 289.087,A -85,B 0,C 180,E1 -21311.713,E2 -21311.713} C_VEL
LIN {X 0,Y 207.172,Z 292.582,A -85,B 0,C 180,E1 -21312.959,E2 -21312.959} C_VEL
LIN {X 0,Y 203.18,Z 297.7,A -85,B 0,C 180,E1 -21315.052,E2 -21315.052} C_VEL
LIN {X 0,Y 199.461,Z 302.168,A -85,B 0,C 180,E1 -21317.339,E2 -21317.339} C_VEL
LIN {X 0,Y 198.365,Z 304.612,A -85,B 0,C 180,E1 -21318.857,E2 -21318.857} C_VEL
LIN {X 0,Y 197.814,Z 308.666,A -85,B 0,C 180,E1 -21321.83,E2 -21321.83} C_VEL
LIN {X 0,Y 197.634,Z 311.59,A -85,B 0,C 180,E1 -21324.694,E2 -21324.694} C_VEL
LIN {X 0,Y 197.633,Z 313.849,A -85,B 0,C 180,E1 -21327.962,E2 -21327.962} C_VEL
LIN {X 0,Y 197.669,Z 314.707,A -85,B 0,C 180,E1 -21330,E2 -21330} C_VEL
LIN {X 0,Y 197.599,Z 315.151,A -85,B 0,C 180,E1 -21332.039,E2 -21332.039} C_VEL
LIN {X 0,Y 197.497,Z 314.766,A -85,B 0,C 180,E1 -21336.129,E2 -21336.129} C_VEL
LIN {X 0,Y 198.029,Z 312.853,A -85,B 0,C 180,E1 -21340.222,E2 -21340.222} C_VEL
LIN {X 0,Y 198.606,Z 311.301,A -85,B 0,C 180,E1 -21342.259,E2 -21342.259} C_VEL
LIN {X 0,Y 199.904,Z 308.194,A -85,B 0,C 180,E1 -21345.289,E2 -21345.289} C_VEL
LIN {X 0,Y 201.894,Z 304.113,A -85,B 0,C 180,E1 -21348.258,E2 -21348.258} C_VEL
LIN {X 0,Y 204.807,Z 297.977,A -85,B 0,C 180,E1 -21351.648,E2 -21351.648} C_VEL
LIN {X 0,Y 208.25,Z 290.168,A -85,B 0,C 180,E1 -21354.952,E2 -21354.952} C_VEL
LIN {X 0,Y 211.966,Z 281.843,A -85,B 0,C 180,E1 -21357.658,E2 -21357.658} C_VEL
LIN {X 0,Y 213.976,Z 276.956,A -85,B 0,C 180,E1 -21358.978,E2 -21358.978} C_VEL
LIN {X 0,Y 216.299,Z 266.697,A -85,B 0,C 180,E1 -21361.649,E2 -21361.649} C_VEL
LIN {X 0,Y 217.285,Z 257.742,A -85,B 0,C 180,E1 -21363.782,E2 -21363.782} C_VEL
LIN {X 0,Y 217.432,Z 247.518,A -85,B 0,C 180,E1 -21366.091,E2 -21366.091} C_VEL
LIN {X 0,Y 216.328,Z 235.726,A -85,B 0,C 180,E1 -21368.765,E2 -21368.765} C_VEL
LIN {X 0,Y 214.288,Z 226.439,A -85,B 0,C 180,E1 -21371.032,E2 -21371.032} C_VEL
LIN {X 0,Y 212.324,Z 221.282,A -85,B 0,C 180,E1 -21372.566,E2 -21372.566} C_VEL
LIN {X 0,Y 210.293,Z 217.275,A -85,B 0,C 180,E1 -21373.972,E2 -21373.972} C_VEL
LIN {X 0,Y 209.609,Z 215.739,A -85,B 0,C 180,E1 -21374.486,E2 -21374.486} C_VEL
LIN {X 0,Y 207.247,Z 211.859,A -85,B 0,C 180,E1 -21376.126,E2 -21376.126} C_VEL
LIN {X 0,Y 206.295,Z 209.594,A -85,B 0,C 180,E1 -21376.888,E2 -21376.888} C_VEL
LIN {X 0,Y 203.564,Z 206.103,A -85,B 0,C 180,E1 -21378.837,E2 -21378.837} C_VEL
LIN {X 0,Y 202.398,Z 203.028,A -85,B 0,C 180,E1 -21379.936,E2 -21379.936} C_VEL
LIN {X 0,Y 202.046,Z 200.753,A -85,B 0,C 180,E1 -21383.747,E2 -21383.747} C_VEL
LIN {X 0,Y 201.643,Z 198.564,A -85,B 0,C 180,E1 -21388.478,E2 -21388.478} C_VEL
LIN {X 0,Y 201.428,Z 196.898,A -85,B 0,C 180,E1 -21393.025,E2 -21393.025} C_VEL
LIN {X 0,Y 201.228,Z 195.716,A -85,B 0,C 180,E1 -21397.406,E2 -21397.406} C_VEL
LIN {X 0,Y 201.156,Z 194.931,A -85,B 0,C 180,E1 -21401.672,E2 -21401.672} C_VEL
LIN {X 0,Y 201.127,Z 194.522,A -85,B 0,C 180,E1 -21405.841,E2 -21405.841} C_VEL
LIN {X 0,Y 201.294,Z 194.411,A -85,B 0,C 180,E1 -21409.945,E2 -21409.945} C_VEL
LIN {X 0,Y 201.361,Z 194.637,A -85,B 0,C 180,E1 -21413.989,E2 -21413.989} C_VEL
LIN {X 0,Y 201.452,Z 194.939,A -85,B 0,C 180,E1 -21414.745,E2 -21414.745} C_VEL
LIN {X 0,Y 202.521,Z 197.248,A -85,B 0,C 180,E1 -21415.832,E2 -21415.832} C_VEL
LIN {X 0,Y 204.932,Z 199.544,A -85,B 0,C 180,E1 -21417.628,E2 -21417.628} C_VEL
LIN {X 0,Y 205.914,Z 200.345,A -85,B 0,C 180,E1 -21418.288,E2 -21418.288} C_VEL
LIN {X 0,Y 208.072,Z 203.914,A -85,B 0,C 180,E1 -21419.999,E2 -21419.999} C_VEL
LIN {X 0,Y 208.977,Z 204.881,A -85,B 0,C 180,E1 -21420.573,E2 -21420.573} C_VEL
LIN {X 0,Y 210.986,Z 208.656,A -85,B 0,C 180,E1 -21422.12,E2 -21422.12} C_VEL
LIN {X 0,Y 214.715,Z 215.74,A -85,B 0,C 180,E1 -21424.88,E2 -21424.88} C_VEL
LIN {X 0,Y 217.047,Z 221.518,A -85,B 0,C 180,E1 -21426.846,E2 -21426.846} C_VEL
LIN {X 0,Y 219.606,Z 230.763,A -85,B 0,C 180,E1 -21429.624,E2 -21429.624} C_VEL
LIN {X 0,Y 220.933,Z 238.783,A -85,B 0,C 180,E1 -21431.932,E2 -21431.932} C_VEL
LIN {X 0,Y 221.288,Z 246.155,A -85,B 0,C 180,E1 -21434.013,E2 -21434.013} C_VEL
LIN {X 0,Y 217.812,Z 255.564,A -85,B 0,C 180,E1 -21436.127,E2 -21436.127} C_VEL
LIN {X 0,Y 214.048,Z 264.461,A -85,B 0,C 180,E1 -21438.636,E2 -21438.636} C_VEL
LIN {X 0,Y 210.841,Z 271.282,A -85,B 0,C 180,E1 -21441.039,E2 -21441.039} C_VEL
LIN {X 0,Y 207.514,Z 277.844,A -85,B 0,C 180,E1 -21443.978,E2 -21443.978} C_VEL
LIN {X 0,Y 204.791,Z 282.756,A -85,B 0,C 180,E1 -21446.839,E2 -21446.839} C_VEL
LIN {X 0,Y 202.504,Z 286.611,A -85,B 0,C 180,E1 -21449.814,E2 -21449.814} C_VEL
LIN {X 0,Y 200.707,Z 289.402,A -85,B 0,C 180,E1 -21452.818,E2 -21452.818} C_VEL
LIN {X 0,Y 198.894,Z 291.639,A -85,B 0,C 180,E1 -21456.919,E2 -21456.919} C_VEL
LIN {X 0,Y 198.116,Z 292.232,A -85,B 0,C 180,E1 -21459.681,E2 -21459.681} C_VEL
LIN {X 0,Y 197.637,Z 292.063,A -85,B 0,C 180,E1 -21462.502,E2 -21462.502} C_VEL
LIN {X 0,Y 197.432,Z 291.096,A -85,B 0,C 180,E1 -21465.392,E2 -21465.392} C_VEL
LIN {X 0,Y 197.55,Z 289.285,A -85,B 0,C 180,E1 -21468.337,E2 -21468.337} C_VEL
LIN {X 0,Y 198.029,Z 286.539,A -85,B 0,C 180,E1 -21471.33,E2 -21471.33} C_VEL
LIN {X 0,Y 198.784,Z 282.676,A -85,B 0,C 180,E1 -21474.404,E2 -21474.404} C_VEL
LIN {X 0,Y 199.878,Z 277.495,A -85,B 0,C 180,E1 -21477.55,E2 -21477.55} C_VEL
LIN {X 0,Y 201.406,Z 270.729,A -85,B 0,C 180,E1 -21480.756,E2 -21480.756} C_VEL
LIN {X 0,Y 203.46,Z 262.179,A -85,B 0,C 180,E1 -21483.907,E2 -21483.907} C_VEL
LIN {X 0,Y 205.449,Z 253.484,A -85,B 0,C 180,E1 -21486.465,E2 -21486.465} C_VEL
LIN {X 0,Y 207.634,Z 243.111,A -85,B 0,C 180,E1 -21488.923,E2 -21488.923} C_VEL
LIN {X 0,Y 209.935,Z 231.107,A -85,B 0,C 180,E1 -21491.139,E2 -21491.139} C_VEL
LIN {X 0,Y 208.184,Z 220.509,A -85,B 0,C 180,E1 -21493.072,E2 -21493.072} C_VEL
LIN {X 0,Y 205.658,Z 208.948,A -85,B 0,C 180,E1 -21494.896,E2 -21494.896} C_VEL
LIN {X 0,Y 201.903,Z 195.451,A -85,B 0,C 180,E1 -21496.711,E2 -21496.711} C_VEL
LIN {X 0,Y 199.32,Z 187.658,A -85,B 0,C 180,E1 -21497.657,E2 -21497.657} C_VEL
LIN {X 0,Y 199.768,Z 187.603,A -85,B 0,C 180,E1 -21500.078,E2 -21500.078} C_VEL
LIN {X 0,Y 199.981,Z 187.576,A -85,B 0,C 180,E1 -21501.919,E2 -21501.919} C_VEL
LIN {X 0,Y 200.318,Z 187.533,A -85,B 0,C 180,E1 -21507.989,E2 -21507.989} C_VEL
LIN {X 0,Y 200.48,Z 187.511,A -85,B 0,C 180,E1 -21510,E2 -21510} C_VEL
LIN {X 0,Y 200.03,Z 187.567,A -85,B 0,C 180,E1 -21514.029,E2 -21514.029} C_VEL
LIN {X 0,Y 200.129,Z 187.559,A -85,B 0,C 180,E1 -21518.075,E2 -21518.075} C_VEL
LIN {X 0,Y 199.912,Z 187.587,A -85,B 0,C 180,E1 -21522.177,E2 -21522.177} C_VEL
LIN {X 0,Y 199.804,Z 187.597,A -85,B 0,C 180,E1 -21526.343,E2 -21526.343} C_VEL
LIN {X 0,Y 199.739,Z 187.607,A -85,B 0,C 180,E1 -21530.601,E2 -21530.601} C_VEL
LIN {X 0,Y 199.673,Z 187.613,A -85,B 0,C 180,E1 -21534.984,E2 -21534.984} C_VEL
LIN {X 0,Y 199.661,Z 187.616,A -85,B 0,C 180,E1 -21539.524,E2 -21539.524} C_VEL
LIN {X 0,Y 199.668,Z 187.613,A -85,B 0,C 180,E1 -21542.356,E2 -21542.356} C_VEL
LIN {X 0,Y 199.62,Z 187.608,A -85,B 0,C 180,E1 -21546.764,E2 -21546.764} C_VEL
LIN {X 0,Y 199.606,Z 187.619,A -85,B 0,C 180,E1 -21549.328,E2 -21549.328} C_VEL
LIN {X 0,Y 199.572,Z 187.624,A -85,B 0,C 180,E1 -21552.311,E2 -21552.311} C_VEL
LIN {X 0,Y 199.578,Z 187.62,A -85,B 0,C 180,E1 -21555.23,E2 -21555.23} C_VEL
LIN {X 0,Y 199.577,Z 187.61,A -85,B 0,C 180,E1 -21558.006,E2 -21558.006} C_VEL
LIN {X 0,Y 199.608,Z 187.614,A -85,B 0,C 180,E1 -21560.768,E2 -21560.768} C_VEL
LIN {X 0,Y 199.61,Z 187.618,A -85,B 0,C 180,E1 -21565.714,E2 -21565.714} C_VEL
LIN {X 0,Y 199.691,Z 187.605,A -85,B 0,C 180,E1 -21568.137,E2 -21568.137} C_VEL
LIN {X 0,Y 199.685,Z 187.601,A -85,B 0,C 180,E1 -21572.773,E2 -21572.773} C_VEL
LIN {X 0,Y 199.749,Z 187.601,A -85,B 0,C 180,E1 -21577.232,E2 -21577.232} C_VEL
LIN {X 0,Y 199.837,Z 187.586,A -85,B 0,C 180,E1 -21581.723,E2 -21581.723} C_VEL
LIN {X 0,Y 199.836,Z 187.58,A -85,B 0,C 180,E1 -21585.749,E2 -21585.749} C_VEL
LIN {X 0,Y 200.022,Z 187.568,A -85,B 0,C 180,E1 -21589.883,E2 -21589.883} C_VEL
LIN {X 0,Y 200.024,Z 187.567,A -85,B 0,C 180,E1 -21593.95,E2 -21593.95} C_VEL
LIN {X 0,Y 200.323,Z 187.519,A -85,B 0,C 180,E1 -21597.99,E2 -21597.99} C_VEL
LIN {X 0,Y 200.48,Z 187.507,A -85,B 0,C 180,E1 -21600.001,E2 -21600.001} C_VEL
LIN {X 0,Y 200.023,Z 187.57,A -85,B 0,C 180,E1 -21604.031,E2 -21604.031} C_VEL
LIN {X 0,Y 200.083,Z 187.552,A -85,B 0,C 180,E1 -21608.078,E2 -21608.078} C_VEL
LIN {X 0,Y 199.876,Z 187.587,A -85,B 0,C 180,E1 -21612.18,E2 -21612.18} C_VEL
LIN {X 0,Y 199.808,Z 187.592,A -85,B 0,C 180,E1 -21616.344,E2 -21616.344} C_VEL
LIN {X 0,Y 199.744,Z 187.602,A -85,B 0,C 180,E1 -21620.602,E2 -21620.602} C_VEL
LIN {X 0,Y 199.678,Z 187.612,A -85,B 0,C 180,E1 -21624.985,E2 -21624.985} C_VEL
LIN {X 0,Y 199.666,Z 187.615,A -85,B 0,C 180,E1 -21629.525,E2 -21629.525} C_VEL
LIN {X 0,Y 199.735,Z 187.752,A -85,B 0,C 180,E1 -21633.998,E2 -21633.998} C_VEL
LIN {X 0,Y 200.252,Z 190.879,A -85,B 0,C 180,E1 -21637.893,E2 -21637.893} C_VEL
LIN {X 0,Y 201.025,Z 195.043,A -85,B 0,C 180,E1 -21642.763,E2 -21642.763} C_VEL
LIN {X 0,Y 201.767,Z 198.906,A -85,B 0,C 180,E1 -21647.012,E2 -21647.012} C_VEL
LIN {X 0,Y 202.27,Z 201.598,A -85,B 0,C 180,E1 -21649.855,E2 -21649.855} C_VEL
LIN {X 0,Y 202.425,Z 203.025,A -85,B 0,C 180,E1 -21651.322,E2 -21651.322} C_VEL
LIN {X 0,Y 202.12,Z 205.539,A -85,B 0,C 180,E1 -21653.764,E2 -21653.764} C_VEL
LIN {X 0,Y 201.187,Z 208.989,A -85,B 0,C 180,E1 -21657.03,E2 -21657.03} C_VEL
LIN {X 0,Y 203.313,Z 221.427,A -85,B 0,C 180,E1 -21658.196,E2 -21658.196} C_VEL
LIN {X 0,Y 204.922,Z 233.538,A -85,B 0,C 180,E1 -21659.616,E2 -21659.616} C_VEL
LIN {X 0,Y 206.132,Z 246.433,A -85,B 0,C 180,E1 -21661.489,E2 -21661.489} C_VEL
LIN {X 0,Y 206.652,Z 257.36,A -85,B 0,C 180,E1 -21663.399,E2 -21663.399} C_VEL
LIN {X 0,Y 206.753,Z 266.972,A -85,B 0,C 180,E1 -21665.392,E2 -21665.392} C_VEL
LIN {X 0,Y 204.506,Z 277.129,A -85,B 0,C 180,E1 -21667.789,E2 -21667.789} C_VEL
LIN {X 0,Y 202.549,Z 285.418,A -85,B 0,C 180,E1 -21670.227,E2 -21670.227} C_VEL
LIN {X 0,Y 200.643,Z 293.546,A -85,B 0,C 180,E1 -21673.204,E2 -21673.204} C_VEL
LIN {X 0,Y 199.328,Z 299.065,A -85,B 0,C 180,E1 -21675.712,E2 -21675.712} C_VEL
LIN {X 0,Y 198.365,Z 304.612,A -85,B 0,C 180,E1 -21678.857,E2 -21678.857} C_VEL
LIN {X 0,Y 197.348,Z 306.863,A -85,B 0,C 180,E1 -21680.421,E2 -21680.421} C_VEL
LIN {X 0,Y 194.126,Z 309.765,A -85,B 0,C 180,E1 -21683.036,E2 -21683.036} C_VEL
LIN {X 0,Y 191.605,Z 311.582,A -85,B 0,C 180,E1 -21685.225,E2 -21685.225} C_VEL
LIN {X 0,Y 190.599,Z 312.724,A -85,B 0,C 180,E1 -21686.95,E2 -21686.95} C_VEL
LIN {X 0,Y 190.546,Z 313.038,A -85,B 0,C 180,E1 -21687.536,E2 -21687.536} C_VEL
LIN {X 0,Y 190.604,Z 314.162,A -85,B 0,C 180,E1 -21690,E2 -21690} C_VEL
LIN {X 0,Y 190.53,Z 314.654,A -85,B 0,C 180,E1 -21692.114,E2 -21692.114} C_VEL
LIN {X 0,Y 190.402,Z 314.682,A -85,B 0,C 180,E1 -21694.711,E2 -21694.711} C_VEL
LIN {X 0,Y 190.617,Z 313.677,A -85,B 0,C 180,E1 -21698.481,E2 -21698.481} C_VEL
LIN {X 0,Y 191.643,Z 311.108,A -85,B 0,C 180,E1 -21702.711,E2 -21702.711} C_VEL
LIN {X 0,Y 193.036,Z 308.102,A -85,B 0,C 180,E1 -21705.847,E2 -21705.847} C_VEL
LIN {X 0,Y 195.136,Z 304.131,A -85,B 0,C 180,E1 -21708.914,E2 -21708.914} C_VEL
LIN {X 0,Y 197.72,Z 299.103,A -85,B 0,C 180,E1 -21711.915,E2 -21711.915} C_VEL
LIN {X 0,Y 201.259,Z 291.747,A -85,B 0,C 180,E1 -21715.327,E2 -21715.327} C_VEL
LIN {X 0,Y 205.05,Z 283.896,A -85,B 0,C 180,E1 -21718.118,E2 -21718.118} C_VEL
LIN {X 0,Y 207.799,Z 277.754,A -85,B 0,C 180,E1 -21719.925,E2 -21719.925} C_VEL
LIN {X 0,Y 210.294,Z 267.82,A -85,B 0,C 180,E1 -21722.645,E2 -21722.645} C_VEL
LIN {X 0,Y 211.57,Z 257.362,A -85,B 0,C 180,E1 -21725.287,E2 -21725.287} C_VEL
LIN {X 0,Y 211.79,Z 248.167,A -85,B 0,C 180,E1 -21727.517,E2 -21727.517} C_VEL
LIN {X 0,Y 211.026,Z 237.94,A -85,B 0,C 180,E1 -21730.003,E2 -21730.003} C_VEL
LIN {X 0,Y 209.73,Z 230.929,A -85,B 0,C 180,E1 -21731.861,E2 -21731.861} C_VEL
LIN {X 0,Y 208.003,Z 226.145,A -85,B 0,C 180,E1 -21733.41,E2 -21733.41} C_VEL
LIN {X 0,Y 206.122,Z 221.563,A -85,B 0,C 180,E1 -21735.063,E2 -21735.063} C_VEL
LIN {X 0,Y 204.218,Z 218.4,A -85,B 0,C 180,E1 -21736.504,E2 -21736.504} C_VEL
LIN {X 0,Y 202.769,Z 215.157,A -85,B 0,C 180,E1 -21737.813,E2 -21737.813} C_VEL
LIN {X 0,Y 200.325,Z 211.3,A -85,B 0,C 180,E1 -21739.901,E2 -21739.901} C_VEL
LIN {X 0,Y 199.389,Z 208.824,A -85,B 0,C 180,E1 -21740.912,E2 -21740.912} C_VEL
LIN {X 0,Y 196.65,Z 205.502,A -85,B 0,C 180,E1 -21743.524,E2 -21743.524} C_VEL
LIN {X 0,Y 195.051,Z 201.858,A -85,B 0,C 180,E1 -21745.624,E2 -21745.624} C_VEL
LIN {X 0,Y 194.925,Z 201.312,A -85,B 0,C 180,E1 -21746.024,E2 -21746.024} C_VEL
LIN {X 0,Y 194.657,Z 199.661,A -85,B 0,C 180,E1 -21750.057,E2 -21750.057} C_VEL
LIN {X 0,Y 194.446,Z 198.176,A -85,B 0,C 180,E1 -21754.636,E2 -21754.636} C_VEL
LIN {X 0,Y 194.28,Z 197.199,A -85,B 0,C 180,E1 -21758.791,E2 -21758.791} C_VEL
LIN {X 0,Y 194.234,Z 196.52,A -85,B 0,C 180,E1 -21763.173,E2 -21763.173} C_VEL
LIN {X 0,Y 194.334,Z 196.162,A -85,B 0,C 180,E1 -21768.553,E2 -21768.553} C_VEL
LIN {X 0,Y 194.402,Z 196.329,A -85,B 0,C 180,E1 -21768.986,E2 -21768.986} C_VEL
LIN {X 0,Y 195.77,Z 198.881,A -85,B 0,C 180,E1 -21770.963,E2 -21770.963} C_VEL
LIN {X 0,Y 198.968,Z 201.553,A -85,B 0,C 180,E1 -21774.17,E2 -21774.17} C_VEL
LIN {X 0,Y 200.522,Z 204.391,A -85,B 0,C 180,E1 -21775.854,E2 -21775.854} C_VEL
LIN {X 0,Y 203.18,Z 207.227,A -85,B 0,C 180,E1 -21778.017,E2 -21778.017} C_VEL
LIN {X 0,Y 205.53,Z 210.812,A -85,B 0,C 180,E1 -21779.999,E2 -21779.999} C_VEL
LIN {X 0,Y 208.948,Z 217.758,A -85,B 0,C 180,E1 -21783.012,E2 -21783.012} C_VEL
LIN {X 0,Y 211.893,Z 224.798,A -85,B 0,C 180,E1 -21785.71,E2 -21785.71} C_VEL
LIN {X 0,Y 214.158,Z 233.993,A -85,B 0,C 180,E1 -21788.719,E2 -21788.719} C_VEL
LIN {X 0,Y 215.27,Z 242.271,A -85,B 0,C 180,E1 -21791.295,E2 -21791.295} C_VEL
LIN {X 0,Y 215.208,Z 248.718,A -85,B 0,C 180,E1 -21793.214,E2 -21793.214} C_VEL
LIN {X 0,Y 211.436,Z 258.027,A -85,B 0,C 180,E1 -21795.431,E2 -21795.431} C_VEL
LIN {X 0,Y 207.189,Z 267.233,A -85,B 0,C 180,E1 -21798.234,E2 -21798.234} C_VEL
LIN {X 0,Y 203.416,Z 274.513,A -85,B 0,C 180,E1 -21801.116,E2 -21801.116} C_VEL
LIN {X 0,Y 200.138,Z 280.339,A -85,B 0,C 180,E1 -21804.074,E2 -21804.074} C_VEL
LIN {X 0,Y 196.945,Z 285.576,A -85,B 0,C 180,E1 -21807.638,E2 -21807.638} C_VEL
LIN {X 0,Y 194.178,Z 289.549,A -85,B 0,C 180,E1 -21811.654,E2 -21811.654} C_VEL
LIN {X 0,Y 192.17,Z 291.941,A -85,B 0,C 180,E1 -21815.812,E2 -21815.812} C_VEL
LIN {X 0,Y 191.073,Z 292.693,A -85,B 0,C 180,E1 -21819.428,E2 -21819.428} C_VEL
LIN {X 0,Y 190.548,Z 292.451,A -85,B 0,C 180,E1 -21822.467,E2 -21822.467} C_VEL
LIN {X 0,Y 190.338,Z 291.39,A -85,B 0,C 180,E1 -21825.448,E2 -21825.448} C_VEL
LIN {X 0,Y 190.456,Z 289.568,A -85,B 0,C 180,E1 -21828.377,E2 -21828.377} C_VEL
LIN {X 0,Y 190.922,Z 286.991,A -85,B 0,C 180,E1 -21831.26,E2 -21831.26} C_VEL
LIN {X 0,Y 191.605,Z 283.683,A -85,B 0,C 180,E1 -21834.064,E2 -21834.064} C_VEL
LIN {X 0,Y 192.811,Z 278.018,A -85,B 0,C 180,E1 -21837.679,E2 -21837.679} C_VEL
LIN {X 0,Y 194.487,Z 270.776,A -85,B 0,C 180,E1 -21841.22,E2 -21841.22} C_VEL
LIN {X 0,Y 196.388,Z 263.109,A -85,B 0,C 180,E1 -21844.142,E2 -21844.142} C_VEL
LIN {X 0,Y 198.7,Z 253.358,A -85,B 0,C 180,E1 -21847.103,E2 -21847.103} C_VEL
LIN {X 0,Y 200.898,Z 243.355,A -85,B 0,C 180,E1 -21849.523,E2 -21849.523} C_VEL
LIN {X 0,Y 203.089,Z 232.514,A -85,B 0,C 180,E1 -21851.599,E2 -21851.599} C_VEL
LIN {X 0,Y 201.959,Z 224.687,A -85,B 0,C 180,E1 -21853.129,E2 -21853.129} C_VEL
LIN {X 0,Y 199.528,Z 212.585,A -85,B 0,C 180,E1 -21855.204,E2 -21855.204} C_VEL
LIN {X 0,Y 196.248,Z 199.928,A -85,B 0,C 180,E1 -21857.066,E2 -21857.066} C_VEL
LIN {X 0,Y 192.429,Z 188.515,A -85,B 0,C 180,E1 -21858.546,E2 -21858.546} C_VEL
LIN {X 0,Y 192.906,Z 188.456,A -85,B 0,C 180,E1 -21861.62,E2 -21861.62} C_VEL
LIN {X 0,Y 193.259,Z 188.412,A -85,B 0,C 180,E1 -21867.916,E2 -21867.916} C_VEL
LIN {X 0,Y 193.444,Z 188.388,A -85,B 0,C 180,E1 -21870,E2 -21870} C_VEL
LIN {X 0,Y 192.977,Z 188.444,A -85,B 0,C 180,E1 -21874.177,E2 -21874.177} C_VEL
LIN {X 0,Y 193.076,Z 188.436,A -85,B 0,C 180,E1 -21878.372,E2 -21878.372} C_VEL
LIN {X 0,Y 192.851,Z 188.465,A -85,B 0,C 180,E1 -21882.63,E2 -21882.63} C_VEL
LIN {X 0,Y 192.779,Z 188.469,A -85,B 0,C 180,E1 -21888.587,E2 -21888.587} C_VEL
LIN {X 0,Y 192.666,Z 188.485,A -85,B 0,C 180,E1 -21894.228,E2 -21894.228} C_VEL
LIN {X 0,Y 192.641,Z 188.487,A -85,B 0,C 180,E1 -21898.889,E2 -21898.889} C_VEL
LIN {X 0,Y 192.593,Z 188.495,A -85,B 0,C 180,E1 -21903.187,E2 -21903.187} C_VEL
LIN {X 0,Y 192.548,Z 188.493,A -85,B 0,C 180,E1 -21908.352,E2 -21908.352} C_VEL
LIN {X 0,Y 192.489,Z 188.508,A -85,B 0,C 180,E1 -21913.097,E2 -21913.097} C_VEL
LIN {X 0,Y 192.489,Z 188.497,A -85,B 0,C 180,E1 -21916.905,E2 -21916.905} C_VEL
LIN {X 0,Y 192.549,Z 188.496,A -85,B 0,C 180,E1 -21921.649,E2 -21921.649} C_VEL
LIN {X 0,Y 192.595,Z 188.492,A -85,B 0,C 180,E1 -21926.815,E2 -21926.815} C_VEL
LIN {X 0,Y 192.659,Z 188.471,A -85,B 0,C 180,E1 -21931.692,E2 -21931.692} C_VEL
LIN {X 0,Y 192.711,Z 188.478,A -85,B 0,C 180,E1 -21936.35,E2 -21936.35} C_VEL
LIN {X 0,Y 192.781,Z 188.464,A -85,B 0,C 180,E1 -21941.414,E2 -21941.414} C_VEL
LIN {X 0,Y 192.764,Z 188.46,A -85,B 0,C 180,E1 -21945.215,E2 -21945.215} C_VEL
LIN {X 0,Y 192.945,Z 188.448,A -85,B 0,C 180,E1 -21949.568,E2 -21949.568} C_VEL
LIN {X 0,Y 192.986,Z 188.444,A -85,B 0,C 180,E1 -21953.729,E2 -21953.729} C_VEL
LIN {X 0,Y 193.265,Z 188.398,A -85,B 0,C 180,E1 -21957.917,E2 -21957.917} C_VEL
LIN {X 0,Y 193.444,Z 188.383,A -85,B 0,C 180,E1 -21960.001,E2 -21960.001} C_VEL
LIN {X 0,Y 192.969,Z 188.448,A -85,B 0,C 180,E1 -21964.178,E2 -21964.178} C_VEL
LIN {X 0,Y 193.032,Z 188.429,A -85,B 0,C 180,E1 -21968.375,E2 -21968.375} C_VEL
LIN {X 0,Y 192.804,Z 188.467,A -85,B 0,C 180,E1 -21972.634,E2 -21972.634} C_VEL
LIN {X 0,Y 192.773,Z 188.468,A -85,B 0,C 180,E1 -21976.958,E2 -21976.958} C_VEL
LIN {X 0,Y 192.67,Z 188.485,A -85,B 0,C 180,E1 -21981.394,E2 -21981.394} C_VEL
LIN {X 0,Y 192.671,Z 188.484,A -85,B 0,C 180,E1 -21984.229,E2 -21984.229} C_VEL
LIN {X 0,Y 192.646,Z 188.489,A -85,B 0,C 180,E1 -21988.89,E2 -21988.89} C_VEL
LIN {X 0,Y 192.669,Z 188.623,A -85,B 0,C 180,E1 -21993.486,E2 -21993.486} C_VEL
LIN {X 0,Y 193.297,Z 192.265,A -85,B 0,C 180,E1 -21998.178,E2 -21998.178} C_VEL
LIN {X 0,Y 194.118,Z 196.807,A -85,B 0,C 180,E1 -22003.607,E2 -22003.607} C_VEL
LIN {X 0,Y 194.871,Z 200.513,A -85,B 0,C 180,E1 -22007.812,E2 -22007.812} C_VEL
LIN {X 0,Y 195.333,Z 203.453,A -85,B 0,C 180,E1 -22010.976,E2 -22010.976} C_VEL
LIN {X 0,Y 195.088,Z 206.003,A -85,B 0,C 180,E1 -22013.566,E2 -22013.566} C_VEL
LIN {X 0,Y 194.355,Z 208.565,A -85,B 0,C 180,E1 -22016.094,E2 -22016.094} C_VEL
LIN {X 0,Y 196.606,Z 221.976,A -85,B 0,C 180,E1 -22017.43,E2 -22017.43} C_VEL
LIN {X 0,Y 198.156,Z 234.214,A -85,B 0,C 180,E1 -22018.965,E2 -22018.965} C_VEL
LIN {X 0,Y 199.258,Z 246.386,A -85,B 0,C 180,E1 -22020.824,E2 -22020.824} C_VEL
LIN {X 0,Y 199.783,Z 258.602,A -85,B 0,C 180,E1 -22023.069,E2 -22023.069} C_VEL
LIN {X 0,Y 199.602,Z 268.653,A -85,B 0,C 180,E1 -22025.284,E2 -22025.284} C_VEL
LIN {X 0,Y 197.122,Z 278.823,A -85,B 0,C 180,E1 -22027.883,E2 -22027.883} C_VEL
LIN {X 0,Y 195.129,Z 287.124,A -85,B 0,C 180,E1 -22030.54,E2 -22030.54} C_VEL
LIN {X 0,Y 193.254,Z 294.82,A -85,B 0,C 180,E1 -22033.63,E2 -22033.63} C_VEL
LIN {X 0,Y 191.668,Z 301.885,A -85,B 0,C 180,E1 -22037.291,E2 -22037.291} C_VEL
LIN {X 0,Y 190.934,Z 306.581,A -85,B 0,C 180,E1 -22040.466,E2 -22040.466} C_VEL
LIN {X 0,Y 190.594,Z 310.134,A -85,B 0,C 180,E1 -22043.649,E2 -22043.649} C_VEL
LIN {X 0,Y 190.535,Z 311.935,A -85,B 0,C 180,E1 -22045.77,E2 -22045.77} C_VEL
LIN {X 0,Y 190.546,Z 313.038,A -85,B 0,C 180,E1 -22047.536,E2 -22047.536} C_VEL
LIN {X 0,Y 189.91,Z 313.925,A -85,B 0,C 180,E1 -22049.28,E2 -22049.28} C_VEL
LIN {X 0,Y 188.276,Z 314.432,A -85,B 0,C 180,E1 -22051.006,E2 -22051.006} C_VEL
LIN {X 0,Y 184.421,Z 314.474,A -85,B 0,C 180,E1 -22054.521,E2 -22054.521} C_VEL
LIN {X 0,Y 183.401,Z 314.095,A -85,B 0,C 180,E1 -22056.365,E2 -22056.365} C_VEL
LIN {X 0,Y 183.352,Z 313.918,A -85,B 0,C 180,E1 -22056.989,E2 -22056.989} C_VEL
LIN {X 0,Y 184.027,Z 312.326,A -85,B 0,C 180,E1 -22061.009,E2 -22061.009} C_VEL
LIN {X 0,Y 185.575,Z 309.096,A -85,B 0,C 180,E1 -22065.373,E2 -22065.373} C_VEL
LIN {X 0,Y 187.61,Z 305.56,A -85,B 0,C 180,E1 -22068.568,E2 -22068.568} C_VEL
LIN {X 0,Y 190.122,Z 301.036,A -85,B 0,C 180,E1 -22071.695,E2 -22071.695} C_VEL
LIN {X 0,Y 193.683,Z 294.472,A -85,B 0,C 180,E1 -22075.18,E2 -22075.18} C_VEL
LIN {X 0,Y 197.446,Z 287.207,A -85,B 0,C 180,E1 -22078.141,E2 -22078.141} C_VEL
LIN {X 0,Y 201.081,Z 280.042,A -85,B 0,C 180,E1 -22080.451,E2 -22080.451} C_VEL
LIN {X 0,Y 203.68,Z 271.748,A -85,B 0,C 180,E1 -22082.92,E2 -22082.92} C_VEL
LIN {X 0,Y 205.271,Z 263.963,A -85,B 0,C 180,E1 -22085.076,E2 -22085.076} C_VEL
LIN {X 0,Y 206.25,Z 253.409,A -85,B 0,C 180,E1 -22087.833,E2 -22087.833} C_VEL
LIN {X 0,Y 206.061,Z 242.706,A -85,B 0,C 180,E1 -22090.634,E2 -22090.634} C_VEL
LIN {X 0,Y 205.147,Z 235.81,A -85,B 0,C 180,E1 -22092.561,E2 -22092.561} C_VEL
LIN {X 0,Y 203.646,Z 230.927,A -85,B 0,C 180,E1 -22094.265,E2 -22094.265} C_VEL
LIN {X 0,Y 202.033,Z 226.711,A -85,B 0,C 180,E1 -22095.913,E2 -22095.913} C_VEL
LIN {X 0,Y 199.857,Z 221.821,A -85,B 0,C 180,E1 -22098.075,E2 -22098.075} C_VEL
LIN {X 0,Y 197.6,Z 218.06,A -85,B 0,C 180,E1 -22100.192,E2 -22100.192} C_VEL
LIN {X 0,Y 196.022,Z 214.494,A -85,B 0,C 180,E1 -22102.072,E2 -22102.072} C_VEL
LIN {X 0,Y 193.346,Z 210.058,A -85,B 0,C 180,E1 -22105.299,E2 -22105.299} C_VEL
LIN {X 0,Y 192.625,Z 207.817,A -85,B 0,C 180,E1 -22106.635,E2 -22106.635} C_VEL
LIN {X 0,Y 189.033,Z 202.861,A -85,B 0,C 180,E1 -22114.237,E2 -22114.237} C_VEL
LIN {X 0,Y 188.66,Z 201.655,A -85,B 0,C 180,E1 -22118.128,E2 -22118.128} C_VEL
LIN {X 0,Y 189.066,Z 201.571,A -85,B 0,C 180,E1 -22121.58,E2 -22121.58} C_VEL
LIN {X 0,Y 192.389,Z 203.092,A -85,B 0,C 180,E1 -22128.522,E2 -22128.522} C_VEL
LIN {X 0,Y 193.832,Z 205.823,A -85,B 0,C 180,E1 -22130.937,E2 -22130.937} C_VEL
LIN {X 0,Y 196.394,Z 208.334,A -85,B 0,C 180,E1 -22133.836,E2 -22133.836} C_VEL
LIN {X 0,Y 198.251,Z 211.323,A -85,B 0,C 180,E1 -22135.933,E2 -22135.933} C_VEL
LIN {X 0,Y 199.284,Z 212.45,A -85,B 0,C 180,E1 -22136.888,E2 -22136.888} C_VEL
LIN {X 0,Y 201.533,Z 216.045,A -85,B 0,C 180,E1 -22139.062,E2 -22139.062} C_VEL
LIN {X 0,Y 204.353,Z 222.094,A -85,B 0,C 180,E1 -22141.97,E2 -22141.97} C_VEL
LIN {X 0,Y 206.58,Z 227.712,A -85,B 0,C 180,E1 -22144.389,E2 -22144.389} C_VEL
LIN {X 0,Y 208.167,Z 234.071,A -85,B 0,C 180,E1 -22146.683,E2 -22146.683} C_VEL
LIN {X 0,Y 209.418,Z 242.79,A -85,B 0,C 180,E1 -22149.659,E2 -22149.659} C_VEL
LIN {X 0,Y 209.468,Z 250.064,A -85,B 0,C 180,E1 -22152.032,E2 -22152.032} C_VEL
LIN {X 0,Y 207.142,Z 255.938,A -85,B 0,C 180,E1 -22153.465,E2 -22153.465} C_VEL
LIN {X 0,Y 202.858,Z 265.004,A -85,B 0,C 180,E1 -22156.09,E2 -22156.09} C_VEL
LIN {X 0,Y 198.549,Z 273.132,A -85,B 0,C 180,E1 -22159.111,E2 -22159.111} C_VEL
LIN {X 0,Y 194.765,Z 279.571,A -85,B 0,C 180,E1 -22162.262,E2 -22162.262} C_VEL
LIN {X 0,Y 191.825,Z 284.08,A -85,B 0,C 180,E1 -22165.125,E2 -22165.125} C_VEL
LIN {X 0,Y 188.773,Z 288.441,A -85,B 0,C 180,E1 -22168.945,E2 -22168.945} C_VEL
LIN {X 0,Y 186.99,Z 290.691,A -85,B 0,C 180,E1 -22171.747,E2 -22171.747} C_VEL
LIN {X 0,Y 185.549,Z 292.211,A -85,B 0,C 180,E1 -22174.62,E2 -22174.62} C_VEL
LIN {X 0,Y 184.481,Z 293.01,A -85,B 0,C 180,E1 -22177.554,E2 -22177.554} C_VEL
LIN {X 0,Y 183.752,Z 293.115,A -85,B 0,C 180,E1 -22180.555,E2 -22180.555} C_VEL
LIN {X 0,Y 183.345,Z 292.462,A -85,B 0,C 180,E1 -22183.627,E2 -22183.627} C_VEL
LIN {X 0,Y 183.243,Z 290.955,A -85,B 0,C 180,E1 -22186.777,E2 -22186.777} C_VEL
LIN {X 0,Y 183.552,Z 288.565,A -85,B 0,C 180,E1 -22189.974,E2 -22189.974} C_VEL
LIN {X 0,Y 184.27,Z 285.18,A -85,B 0,C 180,E1 -22193.217,E2 -22193.217} C_VEL
LIN {X 0,Y 185.24,Z 280.536,A -85,B 0,C 180,E1 -22196.58,E2 -22196.58} C_VEL
LIN {X 0,Y 186.659,Z 274.461,A -85,B 0,C 180,E1 -22199.993,E2 -22199.993} C_VEL
LIN {X 0,Y 188.657,Z 266.527,A -85,B 0,C 180,E1 -22203.446,E2 -22203.446} C_VEL
LIN {X 0,Y 190.942,Z 257.608,A -85,B 0,C 180,E1 -22206.505,E2 -22206.505} C_VEL
LIN {X 0,Y 193.117,Z 248.354,A -85,B 0,C 180,E1 -22209.053,E2 -22209.053} C_VEL
LIN {X 0,Y 195.418,Z 237.704,A -85,B 0,C 180,E1 -22211.386,E2 -22211.386} C_VEL
LIN {X 0,Y 196.299,Z 232.923,A -85,B 0,C 180,E1 -22212.282,E2 -22212.282} C_VEL
LIN {X 0,Y 194.44,Z 221.697,A -85,B 0,C 180,E1 -22214.517,E2 -22214.517} C_VEL
LIN {X 0,Y 191.952,Z 210.155,A -85,B 0,C 180,E1 -22216.502,E2 -22216.502} C_VEL
LIN {X 0,Y 188.424,Z 197.664,A -85,B 0,C 180,E1 -22218.366,E2 -22218.366} C_VEL
LIN {X 0,Y 185.579,Z 189.73,A -85,B 0,C 180,E1 -22219.464,E2 -22219.464} C_VEL
LIN {X 0,Y 185.564,Z 189.37,A -85,B 0,C 180,E1 -22219.539,E2 -22219.539} C_VEL
LIN {X 0,Y 185.805,Z 189.34,A -85,B 0,C 180,E1 -22221.297,E2 -22221.297} C_VEL
LIN {X 0,Y 185.909,Z 189.331,A -85,B 0,C 180,E1 -22225.664,E2 -22225.664} C_VEL
LIN {X 0,Y 186.407,Z 189.264,A -85,B 0,C 180,E1 -22230,E2 -22230} C_VEL
LIN {X 0,Y 185.925,Z 189.322,A -85,B 0,C 180,E1 -22234.335,E2 -22234.335} C_VEL
LIN {X 0,Y 186.026,Z 189.314,A -85,B 0,C 180,E1 -22238.691,E2 -22238.691} C_VEL
LIN {X 0,Y 185.762,Z 189.349,A -85,B 0,C 180,E1 -22243.12,E2 -22243.12} C_VEL
LIN {X 0,Y 185.714,Z 189.349,A -85,B 0,C 180,E1 -22247.622,E2 -22247.622} C_VEL
LIN {X 0,Y 185.613,Z 189.367,A -85,B 0,C 180,E1 -22252.249,E2 -22252.249} C_VEL
LIN {X 0,Y 185.558,Z 189.363,A -85,B 0,C 180,E1 -22257.032,E2 -22257.032} C_VEL
LIN {X 0,Y 185.574,Z 189.37,A -85,B 0,C 180,E1 -22259.494,E2 -22259.494} C_VEL
LIN {X 0,Y 185.495,Z 189.375,A -85,B 0,C 180,E1 -22264.633,E2 -22264.633} C_VEL
LIN {X 0,Y 185.502,Z 189.368,A -85,B 0,C 180,E1 -22267.314,E2 -22267.314} C_VEL
LIN {X 0,Y 185.469,Z 189.381,A -85,B 0,C 180,E1 -22270.726,E2 -22270.726} C_VEL
LIN {X 0,Y 185.459,Z 189.376,A -85,B 0,C 180,E1 -22276.055,E2 -22276.055} C_VEL
LIN {X 0,Y 185.466,Z 189.373,A -85,B 0,C 180,E1 -22279.896,E2 -22279.896} C_VEL
LIN {X 0,Y 185.504,Z 189.376,A -85,B 0,C 180,E1 -22282.712,E2 -22282.712} C_VEL
LIN {X 0,Y 185.54,Z 189.368,A -85,B 0,C 180,E1 -22287.976,E2 -22287.976} C_VEL
LIN {X 0,Y 185.579,Z 189.353,A -85,B 0,C 180,E1 -22290.578,E2 -22290.578} C_VEL
LIN {X 0,Y 185.605,Z 189.361,A -85,B 0,C 180,E1 -22295.386,E2 -22295.386} C_VEL
LIN {X 0,Y 185.71,Z 189.345,A -85,B 0,C 180,E1 -22301.102,E2 -22301.102} C_VEL
LIN {X 0,Y 185.731,Z 189.343,A -85,B 0,C 180,E1 -22306.878,E2 -22306.878} C_VEL
LIN {X 0,Y 185.983,Z 189.317,A -85,B 0,C 180,E1 -22311.307,E2 -22311.307} C_VEL
LIN {X 0,Y 186.208,Z 189.276,A -85,B 0,C 180,E1 -22317.838,E2 -22317.838} C_VEL
LIN {X 0,Y 186.408,Z 189.259,A -85,B 0,C 180,E1 -22320.001,E2 -22320.001} C_VEL
LIN {X 0,Y 185.915,Z 189.326,A -85,B 0,C 180,E1 -22324.337,E2 -22324.337} C_VEL
LIN {X 0,Y 185.98,Z 189.306,A -85,B 0,C 180,E1 -22328.695,E2 -22328.695} C_VEL
LIN {X 0,Y 185.731,Z 189.349,A -85,B 0,C 180,E1 -22333.124,E2 -22333.124} C_VEL
LIN {X 0,Y 185.719,Z 189.344,A -85,B 0,C 180,E1 -22337.623,E2 -22337.623} C_VEL
LIN {X 0,Y 185.618,Z 189.363,A -85,B 0,C 180,E1 -22342.25,E2 -22342.25} C_VEL
LIN {X 0,Y 185.563,Z 189.372,A -85,B 0,C 180,E1 -22347.033,E2 -22347.033} C_VEL
LIN {X 0,Y 185.563,Z 189.371,A -85,B 0,C 180,E1 -22352.023,E2 -22352.023} C_VEL
LIN {X 0,Y 185.593,Z 189.402,A -85,B 0,C 180,E1 -22352.835,E2 -22352.835} C_VEL
LIN {X 0,Y 186.206,Z 192.925,A -85,B 0,C 180,E1 -22357.57,E2 -22357.57} C_VEL
LIN {X 0,Y 186.928,Z 196.941,A -85,B 0,C 180,E1 -22362.592,E2 -22362.592} C_VEL
LIN {X 0,Y 187.79,Z 201.218,A -85,B 0,C 180,E1 -22367.651,E2 -22367.651} C_VEL
LIN {X 0,Y 188.233,Z 203.856,A -85,B 0,C 180,E1 -22370.601,E2 -22370.601} C_VEL
LIN {X 0,Y 188.054,Z 206.386,A -85,B 0,C 180,E1 -22373.277,E2 -22373.277} C_VEL
LIN {X 0,Y 187.538,Z 208.192,A -85,B 0,C 180,E1 -22375.13,E2 -22375.13} C_VEL
LIN {X 0,Y 189.708,Z 221.077,A -85,B 0,C 180,E1 -22376.464,E2 -22376.464} C_VEL
LIN {X 0,Y 191.345,Z 233.804,A -85,B 0,C 180,E1 -22378.113,E2 -22378.113} C_VEL
LIN {X 0,Y 192.387,Z 246.631,A -85,B 0,C 180,E1 -22380.158,E2 -22380.158} C_VEL
LIN {X 0,Y 192.836,Z 257.859,A -85,B 0,C 180,E1 -22382.311,E2 -22382.311} C_VEL
LIN {X 0,Y 192.816,Z 268.032,A -85,B 0,C 180,E1 -22384.642,E2 -22384.642} C_VEL
LIN {X 0,Y 190.423,Z 277.793,A -85,B 0,C 180,E1 -22387.201,E2 -22387.201} C_VEL
LIN {X 0,Y 188.403,Z 285.828,A -85,B 0,C 180,E1 -22389.815,E2 -22389.815} C_VEL
LIN {X 0,Y 186.415,Z 293.726,A -85,B 0,C 180,E1 -22393.012,E2 -22393.012} C_VEL
LIN {X 0,Y 185.084,Z 299.057,A -85,B 0,C 180,E1 -22395.711,E2 -22395.711} C_VEL
LIN {X 0,Y 184.135,Z 304.287,A -85,B 0,C 180,E1 -22398.999,E2 -22398.999} C_VEL
LIN {X 0,Y 183.609,Z 308.315,A -85,B 0,C 180,E1 -22402.301,E2 -22402.301} C_VEL
LIN {X 0,Y 183.457,Z 311.258,A -85,B 0,C 180,E1 -22405.606,E2 -22405.606} C_VEL
LIN {X 0,Y 183.507,Z 312.665,A -85,B 0,C 180,E1 -22407.806,E2 -22407.806} C_VEL
LIN {X 0,Y 183.539,Z 313.616,A -85,B 0,C 180,E1 -22410,E2 -22410} C_VEL
LIN {X 0,Y 183.462,Z 314.153,A -85,B 0,C 180,E1 -22412.196,E2 -22412.196} C_VEL
LIN {X 0,Y 183.327,Z 314.291,A -85,B 0,C 180,E1 -22414.621,E2 -22414.621} C_VEL
LIN {X 0,Y 183.352,Z 313.918,A -85,B 0,C 180,E1 -22416.989,E2 -22416.989} C_VEL
LIN {X 0,Y 182.869,Z 313.347,A -85,B 0,C 180,E1 -22418.822,E2 -22418.822} C_VEL
LIN {X 0,Y 180.601,Z 311.858,A -85,B 0,C 180,E1 -22421.836,E2 -22421.836} C_VEL
LIN {X 0,Y 178.833,Z 309.844,A -85,B 0,C 180,E1 -22424.884,E2 -22424.884} C_VEL
LIN {X 0,Y 179.137,Z 308.287,A -85,B 0,C 180,E1 -22426.709,E2 -22426.709} C_VEL
LIN {X 0,Y 181.681,Z 304.226,A -85,B 0,C 180,E1 -22430.375,E2 -22430.375} C_VEL
LIN {X 0,Y 184.623,Z 299.489,A -85,B 0,C 180,E1 -22433.56,E2 -22433.56} C_VEL
LIN {X 0,Y 188.537,Z 292.5,A -85,B 0,C 180,E1 -22437.171,E2 -22437.171} C_VEL
LIN {X 0,Y 192.709,Z 285.088,A -85,B 0,C 180,E1 -22440.097,E2 -22440.097} C_VEL
LIN {X 0,Y 195.636,Z 279.27,A -85,B 0,C 180,E1 -22441.998,E2 -22441.998} C_VEL
LIN {X 0,Y 198.257,Z 271.034,A -85,B 0,C 180,E1 -22444.555,E2 -22444.555} C_VEL
LIN {X 0,Y 199.993,Z 261.909,A -85,B 0,C 180,E1 -22447.19,E2 -22447.19} C_VEL
LIN {X 0,Y 200.793,Z 254.204,A -85,B 0,C 180,E1 -22449.357,E2 -22449.357} C_VEL
LIN {X 0,Y 200.847,Z 244.743,A -85,B 0,C 180,E1 -22452.007,E2 -22452.007} C_VEL
LIN {X 0,Y 200.434,Z 240.313,A -85,B 0,C 180,E1 -22453.353,E2 -22453.353} C_VEL
LIN {X 0,Y 199.178,Z 235.65,A -85,B 0,C 180,E1 -22455.112,E2 -22455.112} C_VEL
LIN {X 0,Y 197.824,Z 231.721,A -85,B 0,C 180,E1 -22456.762,E2 -22456.762} C_VEL
LIN {X 0,Y 196.169,Z 227.385,A -85,B 0,C 180,E1 -22458.795,E2 -22458.795} C_VEL
LIN {X 0,Y 193.815,Z 222.499,A -85,B 0,C 180,E1 -22461.561,E2 -22461.561} C_VEL
LIN {X 0,Y 193.204,Z 220.932,A -85,B 0,C 180,E1 -22462.462,E2 -22462.462} C_VEL
LIN {X 0,Y 191.092,Z 217.291,A -85,B 0,C 180,E1 -22465.244,E2 -22465.244} C_VEL
LIN {X 0,Y 189.737,Z 213.839,A -85,B 0,C 180,E1 -22467.87,E2 -22467.87} C_VEL
LIN {X 0,Y 187.15,Z 209.58,A -85,B 0,C 180,E1 -22474.622,E2 -22474.622} C_VEL
LIN {X 0,Y 186.861,Z 208.565,A -85,B 0,C 180,E1 -22477.906,E2 -22477.906} C_VEL
LIN {X 0,Y 187.19,Z 208.411,A -85,B 0,C 180,E1 -22481.389,E2 -22481.389} C_VEL
LIN {X 0,Y 189.472,Z 209.528,A -85,B 0,C 180,E1 -22487.14,E2 -22487.14} C_VEL
LIN {X 0,Y 192.874,Z 214.066,A -85,B 0,C 180,E1 -22492.672,E2 -22492.672} C_VEL
LIN {X 0,Y 196.963,Z 220.256,A -85,B 0,C 180,E1 -22497.571,E2 -22497.571} C_VEL
LIN {X 0,Y 199.835,Z 226.553,A -85,B 0,C 180,E1 -22501.007,E2 -22501.007} C_VEL
LIN {X 0,Y 202.047,Z 233.12,A -85,B 0,C 180,E1 -22503.988,E2 -22503.988} C_VEL
LIN {X 0,Y 203.392,Z 240.864,A -85,B 0,C 180,E1 -22506.945,E2 -22506.945} C_VEL
LIN {X 0,Y 203.838,Z 247.687,A -85,B 0,C 180,E1 -22509.425,E2 -22509.425} C_VEL
LIN {X 0,Y 203.723,Z 252.001,A -85,B 0,C 180,E1 -22510.936,E2 -22510.936} C_VEL
LIN {X 0,Y 202.034,Z 256.256,A -85,B 0,C 180,E1 -22512.046,E2 -22512.046} C_VEL
LIN {X 0,Y 198.015,Z 264.373,A -85,B 0,C 180,E1 -22514.384,E2 -22514.384} C_VEL
LIN {X 0,Y 193.278,Z 272.778,A -85,B 0,C 180,E1 -22517.497,E2 -22517.497} C_VEL
LIN {X 0,Y 189.656,Z 278.646,A -85,B 0,C 180,E1 -22520.3,E2 -22520.3} C_VEL
LIN {X 0,Y 186.411,Z 283.394,A -85,B 0,C 180,E1 -22523.185,E2 -22523.185} C_VEL
LIN {X 0,Y 183.75,Z 287.059,A -85,B 0,C 180,E1 -22526.093,E2 -22526.093} C_VEL
LIN {X 0,Y 180.599,Z 290.854,A -85,B 0,C 180,E1 -22530.389,E2 -22530.389} C_VEL
LIN {X 0,Y 178.578,Z 292.84,A -85,B 0,C 180,E1 -22534.262,E2 -22534.262} C_VEL
LIN {X 0,Y 177.37,Z 293.574,A -85,B 0,C 180,E1 -22537.582,E2 -22537.582} C_VEL
LIN {X 0,Y 176.591,Z 293.46,A -85,B 0,C 180,E1 -22540.872,E2 -22540.872} C_VEL
LIN {X 0,Y 176.209,Z 292.559,A -85,B 0,C 180,E1 -22544.116,E2 -22544.116} C_VEL
LIN {X 0,Y 176.19,Z 290.908,A -85,B 0,C 180,E1 -22547.303,E2 -22547.303} C_VEL
LIN {X 0,Y 176.782,Z 287.37,A -85,B 0,C 180,E1 -22551.589,E2 -22551.589} C_VEL
LIN {X 0,Y 177.605,Z 283.565,A -85,B 0,C 180,E1 -22554.863,E2 -22554.863} C_VEL
LIN {X 0,Y 178.934,Z 277.836,A -85,B 0,C 180,E1 -22558.639,E2 -22558.639} C_VEL
LIN {X 0,Y 180.647,Z 270.881,A -85,B 0,C 180,E1 -22562.169,E2 -22562.169} C_VEL
LIN {X 0,Y 182.797,Z 262.785,A -85,B 0,C 180,E1 -22565.399,E2 -22565.399} C_VEL
LIN {X 0,Y 185.086,Z 253.805,A -85,B 0,C 180,E1 -22568.271,E2 -22568.271} C_VEL
LIN {X 0,Y 187.467,Z 243.701,A -85,B 0,C 180,E1 -22570.85,E2 -22570.85} C_VEL
LIN {X 0,Y 189.425,Z 234.597,A -85,B 0,C 180,E1 -22572.733,E2 -22572.733} C_VEL
LIN {X 0,Y 188.259,Z 225.939,A -85,B 0,C 180,E1 -22574.574,E2 -22574.574} C_VEL
LIN {X 0,Y 186.078,Z 214.974,A -85,B 0,C 180,E1 -22576.647,E2 -22576.647} C_VEL
LIN {X 0,Y 183.217,Z 203.709,A -85,B 0,C 180,E1 -22578.522,E2 -22578.522} C_VEL
LIN {X 0,Y 179.781,Z 193.686,A -85,B 0,C 180,E1 -22580.047,E2 -22580.047} C_VEL
LIN {X 0,Y 178.666,Z 190.23,A -85,B 0,C 180,E1 -22580.56,E2 -22580.56} C_VEL
LIN {X 0,Y 178.849,Z 190.209,A -85,B 0,C 180,E1 -22583.229,E2 -22583.229} C_VEL
LIN {X 0,Y 179.148,Z 190.169,A -85,B 0,C 180,E1 -22587.751,E2 -22587.751} C_VEL
LIN {X 0,Y 179.37,Z 190.14,A -85,B 0,C 180,E1 -22590,E2 -22590} C_VEL
LIN {X 0,Y 178.873,Z 190.2,A -85,B 0,C 180,E1 -22594.507,E2 -22594.507} C_VEL
LIN {X 0,Y 178.976,Z 190.193,A -85,B 0,C 180,E1 -22599.037,E2 -22599.037} C_VEL
LIN {X 0,Y 178.686,Z 190.233,A -85,B 0,C 180,E1 -22603.65,E2 -22603.65} C_VEL
LIN {X 0,Y 178.677,Z 190.226,A -85,B 0,C 180,E1 -22608.34,E2 -22608.34} C_VEL
LIN {X 0,Y 178.528,Z 190.251,A -85,B 0,C 180,E1 -22613.182,E2 -22613.182} C_VEL
LIN {X 0,Y 178.483,Z 190.25,A -85,B 0,C 180,E1 -22618.197,E2 -22618.197} C_VEL
LIN {X 0,Y 178.474,Z 190.254,A -85,B 0,C 180,E1 -22620.791,E2 -22620.791} C_VEL
LIN {X 0,Y 178.481,Z 190.248,A -85,B 0,C 180,E1 -22624.219,E2 -22624.219} C_VEL
LIN {X 0,Y 178.393,Z 190.259,A -85,B 0,C 180,E1 -22629.075,E2 -22629.075} C_VEL
LIN {X 0,Y 178.396,Z 190.262,A -85,B 0,C 180,E1 -22632.045,E2 -22632.045} C_VEL
LIN {X 0,Y 178.392,Z 190.258,A -85,B 0,C 180,E1 -22635.164,E2 -22635.164} C_VEL
LIN {X 0,Y 178.401,Z 190.246,A -85,B 0,C 180,E1 -22638.46,E2 -22638.46} C_VEL
LIN {X 0,Y 178.42,Z 190.258,A -85,B 0,C 180,E1 -22643.784,E2 -22643.784} C_VEL
LIN {X 0,Y 178.483,Z 190.251,A -85,B 0,C 180,E1 -22646.548,E2 -22646.548} C_VEL
LIN {X 0,Y 178.52,Z 190.235,A -85,B 0,C 180,E1 -22650.008,E2 -22650.008} C_VEL
LIN {X 0,Y 178.533,Z 190.242,A -85,B 0,C 180,E1 -22654.877,E2 -22654.877} C_VEL
LIN {X 0,Y 178.654,Z 190.225,A -85,B 0,C 180,E1 -22660.756,E2 -22660.756} C_VEL
LIN {X 0,Y 178.66,Z 190.219,A -85,B 0,C 180,E1 -22666.349,E2 -22666.349} C_VEL
LIN {X 0,Y 178.912,Z 190.198,A -85,B 0,C 180,E1 -22670.961,E2 -22670.961} C_VEL
LIN {X 0,Y 179.154,Z 190.153,A -85,B 0,C 180,E1 -22677.753,E2 -22677.753} C_VEL
LIN {X 0,Y 179.371,Z 190.135,A -85,B 0,C 180,E1 -22680.001,E2 -22680.001} C_VEL
LIN {X 0,Y 178.863,Z 190.204,A -85,B 0,C 180,E1 -22684.508,E2 -22684.508} C_VEL
LIN {X 0,Y 178.909,Z 190.186,A -85,B 0,C 180,E1 -22689.041,E2 -22689.041} C_VEL
LIN {X 0,Y 178.666,Z 190.231,A -85,B 0,C 180,E1 -22693.653,E2 -22693.653} C_VEL
LIN {X 0,Y 178.682,Z 190.22,A -85,B 0,C 180,E1 -22698.341,E2 -22698.341} C_VEL
LIN {X 0,Y 178.532,Z 190.246,A -85,B 0,C 180,E1 -22703.183,E2 -22703.183} C_VEL
LIN {X 0,Y 178.488,Z 190.253,A -85,B 0,C 180,E1 -22708.198,E2 -22708.198} C_VEL
LIN {X 0,Y 178.537,Z 190.367,A -85,B 0,C 180,E1 -22712.436,E2 -22712.436} C_VEL
LIN {X 0,Y 178.988,Z 192.965,A -85,B 0,C 180,E1 -22716.086,E2 -22716.086} C_VEL
LIN {X 0,Y 179.526,Z 196.08,A -85,B 0,C 180,E1 -22720.237,E2 -22720.237} C_VEL
LIN {X 0,Y 180.338,Z 200.229,A -85,B 0,C 180,E1 -22725.454,E2 -22725.454} C_VEL
LIN {X 0,Y 180.898,Z 202.921,A -85,B 0,C 180,E1 -22728.665,E2 -22728.665} C_VEL
LIN {X 0,Y 181.159,Z 205.528,A -85,B 0,C 180,E1 -22731.632,E2 -22731.632} C_VEL
LIN {X 0,Y 180.761,Z 208.004,A -85,B 0,C 180,E1 -22734.133,E2 -22734.133} C_VEL
LIN {X 0,Y 183.047,Z 221.696,A -85,B 0,C 180,E1 -22735.634,E2 -22735.634} C_VEL
LIN {X 0,Y 184.576,Z 233.798,A -85,B 0,C 180,E1 -22737.299,E2 -22737.299} C_VEL
LIN {X 0,Y 185.521,Z 246.331,A -85,B 0,C 180,E1 -22739.369,E2 -22739.369} C_VEL
LIN {X 0,Y 185.959,Z 257.081,A -85,B 0,C 180,E1 -22741.501,E2 -22741.501} C_VEL
LIN {X 0,Y 185.888,Z 267.368,A -85,B 0,C 180,E1 -22743.927,E2 -22743.927} C_VEL
LIN {X 0,Y 185.288,Z 270.578,A -85,B 0,C 180,E1 -22744.741,E2 -22744.741} C_VEL
LIN {X 0,Y 182.876,Z 279.796,A -85,B 0,C 180,E1 -22747.4,E2 -22747.4} C_VEL
LIN {X 0,Y 180.542,Z 288.764,A -85,B 0,C 180,E1 -22750.678,E2 -22750.678} C_VEL
LIN {X 0,Y 178.697,Z 295.982,A -85,B 0,C 180,E1 -22754.02,E2 -22754.02} C_VEL
LIN {X 0,Y 177.419,Z 301.753,A -85,B 0,C 180,E1 -22757.416,E2 -22757.416} C_VEL
LIN {X 0,Y 176.696,Z 306.274,A -85,B 0,C 180,E1 -22760.846,E2 -22760.846} C_VEL
LIN {X 0,Y 176.422,Z 310.095,A -85,B 0,C 180,E1 -22764.827,E2 -22764.827} C_VEL
LIN {X 0,Y 176.445,Z 312.038,A -85,B 0,C 180,E1 -22767.718,E2 -22767.718} C_VEL
LIN {X 0,Y 176.476,Z 313.057,A -85,B 0,C 180,E1 -22770,E2 -22770} C_VEL
LIN {X 0,Y 176.37,Z 313.641,A -85,B 0,C 180,E1 -22772.284,E2 -22772.284} C_VEL
LIN {X 0,Y 176.265,Z 313.829,A -85,B 0,C 180,E1 -22774.574,E2 -22774.574} C_VEL
LIN {X 0,Y 176.542,Z 313.06,A -85,B 0,C 180,E1 -22779.163,E2 -22779.163} C_VEL
LIN {X 0,Y 177.741,Z 310.703,A -85,B 0,C 180,E1 -22783.724,E2 -22783.724} C_VEL
LIN {X 0,Y 179.137,Z 308.287,A -85,B 0,C 180,E1 -22786.709,E2 -22786.709} C_VEL
LIN {X 0,Y 179.641,Z 306.562,A -85,B 0,C 180,E1 -22788.507,E2 -22788.507} C_VEL
LIN {X 0,Y 179.027,Z 303.367,A -85,B 0,C 180,E1 -22791.5,E2 -22791.5} C_VEL
LIN {X 0,Y 178.769,Z 299.591,A -85,B 0,C 180,E1 -22794.44,E2 -22794.44} C_VEL
LIN {X 0,Y 179.806,Z 296.954,A -85,B 0,C 180,E1 -22796.1,E2 -22796.1} C_VEL
LIN {X 0,Y 183.651,Z 290.712,A -85,B 0,C 180,E1 -22799.204,E2 -22799.204} C_VEL
LIN {X 0,Y 188.271,Z 282.984,A -85,B 0,C 180,E1 -22802.137,E2 -22802.137} C_VEL
LIN {X 0,Y 190.821,Z 277.028,A -85,B 0,C 180,E1 -22804.171,E2 -22804.171} C_VEL
LIN {X 0,Y 193.215,Z 269.18,A -85,B 0,C 180,E1 -22806.679,E2 -22806.679} C_VEL
LIN {X 0,Y 194.949,Z 260.189,A -85,B 0,C 180,E1 -22809.405,E2 -22809.405} C_VEL
LIN {X 0,Y 195.743,Z 249.929,A -85,B 0,C 180,E1 -22812.491,E2 -22812.491} C_VEL
LIN {X 0,Y 195.635,Z 244.998,A -85,B 0,C 180,E1 -22814.069,E2 -22814.069} C_VEL
LIN {X 0,Y 194.61,Z 240.249,A -85,B 0,C 180,E1 -22815.958,E2 -22815.958} C_VEL
LIN {X 0,Y 192.591,Z 234.053,A -85,B 0,C 180,E1 -22818.938,E2 -22818.938} C_VEL
LIN {X 0,Y 191.525,Z 231.429,A -85,B 0,C 180,E1 -22820.408,E2 -22820.408} C_VEL
LIN {X 0,Y 189.956,Z 227.001,A -85,B 0,C 180,E1 -22822.986,E2 -22822.986} C_VEL
LIN {X 0,Y 187.104,Z 220.315,A -85,B 0,C 180,E1 -22828.272,E2 -22828.272} C_VEL
LIN {X 0,Y 185.28,Z 217.273,A -85,B 0,C 180,E1 -22832.922,E2 -22832.922} C_VEL
LIN {X 0,Y 184.723,Z 215.373,A -85,B 0,C 180,E1 -22837.637,E2 -22837.637} C_VEL
LIN {X 0,Y 185.235,Z 215.29,A -85,B 0,C 180,E1 -22842.329,E2 -22842.329} C_VEL
LIN {X 0,Y 187.009,Z 216.185,A -85,B 0,C 180,E1 -22846.967,E2 -22846.967} C_VEL
LIN {X 0,Y 190.014,Z 220.621,A -85,B 0,C 180,E1 -22852.561,E2 -22852.561} C_VEL
LIN {X 0,Y 193.096,Z 225.748,A -85,B 0,C 180,E1 -22856.869,E2 -22856.869} C_VEL
LIN {X 0,Y 195.228,Z 231.083,A -85,B 0,C 180,E1 -22859.999,E2 -22859.999} C_VEL
LIN {X 0,Y 197.056,Z 237.069,A -85,B 0,C 180,E1 -22863.002,E2 -22863.002} C_VEL
LIN {X 0,Y 197.928,Z 243.225,A -85,B 0,C 180,E1 -22865.603,E2 -22865.603} C_VEL
LIN {X 0,Y 198.201,Z 251.047,A -85,B 0,C 180,E1 -22868.666,E2 -22868.666} C_VEL
LIN {X 0,Y 198.056,Z 253.751,A -85,B 0,C 180,E1 -22869.703,E2 -22869.703} C_VEL
LIN {X 0,Y 197.626,Z 255.384,A -85,B 0,C 180,E1 -22870.241,E2 -22870.241} C_VEL
LIN {X 0,Y 193.359,Z 263.7,A -85,B 0,C 180,E1 -22872.595,E2 -22872.595} C_VEL
LIN {X 0,Y 188.347,Z 272.267,A -85,B 0,C 180,E1 -22875.693,E2 -22875.693} C_VEL
LIN {X 0,Y 183.69,Z 279.337,A -85,B 0,C 180,E1 -22879.105,E2 -22879.105} C_VEL
LIN {X 0,Y 180.191,Z 284.067,A -85,B 0,C 180,E1 -22882.101,E2 -22882.101} C_VEL
LIN {X 0,Y 176.605,Z 288.574,A -85,B 0,C 180,E1 -22885.959,E2 -22885.959} C_VEL
LIN {X 0,Y 174.37,Z 290.997,A -85,B 0,C 180,E1 -22888.923,E2 -22888.923} C_VEL
LIN {X 0,Y 172.52,Z 292.73,A -85,B 0,C 180,E1 -22891.976,E2 -22891.976} C_VEL
LIN {X 0,Y 171.094,Z 293.773,A -85,B 0,C 180,E1 -22895.103,E2 -22895.103} C_VEL
LIN {X 0,Y 170.063,Z 294.073,A -85,B 0,C 180,E1 -22898.306,E2 -22898.306} C_VEL
LIN {X 0,Y 169.373,Z 293.643,A -85,B 0,C 180,E1 -22901.677,E2 -22901.677} C_VEL
LIN {X 0,Y 169.06,Z 292.444,A -85,B 0,C 180,E1 -22905.032,E2 -22905.032} C_VEL
LIN {X 0,Y 169.175,Z 290.431,A -85,B 0,C 180,E1 -22908.396,E2 -22908.396} C_VEL
LIN {X 0,Y 169.737,Z 287.428,A -85,B 0,C 180,E1 -22911.876,E2 -22911.876} C_VEL
LIN {X 0,Y 170.649,Z 283.299,A -85,B 0,C 180,E1 -22915.452,E2 -22915.452} C_VEL
LIN {X 0,Y 171.984,Z 277.821,A -85,B 0,C 180,E1 -22919.107,E2 -22919.107} C_VEL
LIN {X 0,Y 173.81,Z 270.647,A -85,B 0,C 180,E1 -22922.816,E2 -22922.816} C_VEL
LIN {X 0,Y 175.811,Z 263.37,A -85,B 0,C 180,E1 -22925.812,E2 -22925.812} C_VEL
LIN {X 0,Y 178.292,Z 253.995,A -85,B 0,C 180,E1 -22928.918,E2 -22928.918} C_VEL
LIN {X 0,Y 180.79,Z 243.756,A -85,B 0,C 180,E1 -22931.6,E2 -22931.6} C_VEL
LIN {X 0,Y 182.693,Z 234.777,A -85,B 0,C 180,E1 -22933.518,E2 -22933.518} C_VEL
LIN {X 0,Y 180.686,Z 222.432,A -85,B 0,C 180,E1 -22936.217,E2 -22936.217} C_VEL
LIN {X 0,Y 178.226,Z 211.044,A -85,B 0,C 180,E1 -22938.355,E2 -22938.355} C_VEL
LIN {X 0,Y 174.956,Z 200.087,A -85,B 0,C 180,E1 -22940.21,E2 -22940.21} C_VEL
LIN {X 0,Y 171.783,Z 191.7,A -85,B 0,C 180,E1 -22941.545,E2 -22941.545} C_VEL
LIN {X 0,Y 171.699,Z 191.098,A -85,B 0,C 180,E1 -22941.689,E2 -22941.689} C_VEL
LIN {X 0,Y 172.094,Z 191.047,A -85,B 0,C 180,E1 -22947.659,E2 -22947.659} C_VEL
LIN {X 0,Y 172.332,Z 191.017,A -85,B 0,C 180,E1 -22950,E2 -22950} C_VEL
LIN {X 0,Y 171.823,Z 191.077,A -85,B 0,C 180,E1 -22954.692,E2 -22954.692} C_VEL
LIN {X 0,Y 171.907,Z 191.073,A -85,B 0,C 180,E1 -22959.411,E2 -22959.411} C_VEL
LIN {X 0,Y 171.61,Z 191.114,A -85,B 0,C 180,E1 -22964.224,E2 -22964.224} C_VEL
LIN {X 0,Y 171.572,Z 191.114,A -85,B 0,C 180,E1 -22969.591,E2 -22969.591} C_VEL
LIN {X 0,Y 171.466,Z 191.119,A -85,B 0,C 180,E1 -22975.616,E2 -22975.616} C_VEL
LIN {X 0,Y 171.437,Z 191.131,A -85,B 0,C 180,E1 -22980.586,E2 -22980.586} C_VEL
LIN {X 0,Y 171.389,Z 191.127,A -85,B 0,C 180,E1 -22985.035,E2 -22985.035} C_VEL
LIN {X 0,Y 171.355,Z 191.134,A -85,B 0,C 180,E1 -22988.808,E2 -22988.808} C_VEL
LIN {X 0,Y 171.319,Z 191.142,A -85,B 0,C 180,E1 -22994.218,E2 -22994.218} C_VEL
LIN {X 0,Y 171.333,Z 191.128,A -85,B 0,C 180,E1 -22998.983,E2 -22998.983} C_VEL
LIN {X 0,Y 171.385,Z 191.132,A -85,B 0,C 180,E1 -23002.042,E2 -23002.042} C_VEL
LIN {X 0,Y 171.396,Z 191.134,A -85,B 0,C 180,E1 -23005.093,E2 -23005.093} C_VEL
LIN {X 0,Y 171.446,Z 191.112,A -85,B 0,C 180,E1 -23010.535,E2 -23010.535} C_VEL
LIN {X 0,Y 171.465,Z 191.122,A -85,B 0,C 180,E1 -23015.804,E2 -23015.804} C_VEL
LIN {X 0,Y 171.61,Z 191.102,A -85,B 0,C 180,E1 -23020.877,E2 -23020.877} C_VEL
LIN {X 0,Y 171.58,Z 191.097,A -85,B 0,C 180,E1 -23025.774,E2 -23025.774} C_VEL
LIN {X 0,Y 171.848,Z 191.079,A -85,B 0,C 180,E1 -23030.586,E2 -23030.586} C_VEL
LIN {X 0,Y 171.817,Z 191.075,A -85,B 0,C 180,E1 -23035.309,E2 -23035.309} C_VEL
LIN {X 0,Y 172.333,Z 191.011,A -85,B 0,C 180,E1 -23040.001,E2 -23040.001} C_VEL
LIN {X 0,Y 171.811,Z 191.082,A -85,B 0,C 180,E1 -23044.694,E2 -23044.694} C_VEL
LIN {X 0,Y 171.847,Z 191.067,A -85,B 0,C 180,E1 -23049.416,E2 -23049.416} C_VEL
LIN {X 0,Y 171.596,Z 191.11,A -85,B 0,C 180,E1 -23054.227,E2 -23054.227} C_VEL
LIN {X 0,Y 171.612,Z 191.101,A -85,B 0,C 180,E1 -23059.126,E2 -23059.126} C_VEL
LIN {X 0,Y 171.471,Z 191.128,A -85,B 0,C 180,E1 -23065.617,E2 -23065.617} C_VEL
LIN {X 0,Y 171.481,Z 191.126,A -85,B 0,C 180,E1 -23071.682,E2 -23071.682} C_VEL
LIN {X 0,Y 171.877,Z 193.444,A -85,B 0,C 180,E1 -23075.136,E2 -23075.136} C_VEL
LIN {X 0,Y 172.573,Z 197.427,A -85,B 0,C 180,E1 -23080.664,E2 -23080.664} C_VEL
LIN {X 0,Y 173.244,Z 200.778,A -85,B 0,C 180,E1 -23085.051,E2 -23085.051} C_VEL
LIN {X 0,Y 173.94,Z 204.577,A -85,B 0,C 180,E1 -23089.724,E2 -23089.724} C_VEL
LIN {X 0,Y 174.093,Z 206.038,A -85,B 0,C 180,E1 -23091.455,E2 -23091.455} C_VEL
LIN {X 0,Y 173.921,Z 207.37,A -85,B 0,C 180,E1 -23092.979,E2 -23092.979} C_VEL
LIN {X 0,Y 176.21,Z 220.723,A -85,B 0,C 180,E1 -23094.536,E2 -23094.536} C_VEL
LIN {X 0,Y 177.783,Z 233.655,A -85,B 0,C 180,E1 -23096.397,E2 -23096.397} C_VEL
LIN {X 0,Y 178.712,Z 246.364,A -85,B 0,C 180,E1 -23098.605,E2 -23098.605} C_VEL
LIN {X 0,Y 179.057,Z 256.826,A -85,B 0,C 180,E1 -23100.778,E2 -23100.778} C_VEL
LIN {X 0,Y 178.95,Z 267.68,A -85,B 0,C 180,E1 -23103.466,E2 -23103.466} C_VEL
LIN {X 0,Y 176.769,Z 276.682,A -85,B 0,C 180,E1 -23106.014,E2 -23106.014} C_VEL
LIN {X 0,Y 174.209,Z 286.074,A -85,B 0,C 180,E1 -23109.33,E2 -23109.33} C_VEL
LIN {X 0,Y 172.158,Z 293.707,A -85,B 0,C 180,E1 -23112.785,E2 -23112.785} C_VEL
LIN {X 0,Y 170.475,Z 300.732,A -85,B 0,C 180,E1 -23116.895,E2 -23116.895} C_VEL
LIN {X 0,Y 169.686,Z 305.387,A -85,B 0,C 180,E1 -23120.464,E2 -23120.464} C_VEL
LIN {X 0,Y 169.359,Z 309.547,A -85,B 0,C 180,E1 -23124.851,E2 -23124.851} C_VEL
LIN {X 0,Y 169.383,Z 311.371,A -85,B 0,C 180,E1 -23127.622,E2 -23127.622} C_VEL
LIN {X 0,Y 169.413,Z 312.483,A -85,B 0,C 180,E1 -23130,E2 -23130} C_VEL
LIN {X 0,Y 169.284,Z 313.129,A -85,B 0,C 180,E1 -23132.38,E2 -23132.38} C_VEL
LIN {X 0,Y 169.177,Z 313.368,A -85,B 0,C 180,E1 -23134.766,E2 -23134.766} C_VEL
LIN {X 0,Y 169.507,Z 312.715,A -85,B 0,C 180,E1 -23139.547,E2 -23139.547} C_VEL
LIN {X 0,Y 170.04,Z 311.828,A -85,B 0,C 180,E1 -23141.927,E2 -23141.927} C_VEL
LIN {X 0,Y 171.871,Z 308.847,A -85,B 0,C 180,E1 -23146.633,E2 -23146.633} C_VEL
LIN {X 0,Y 175.008,Z 304.291,A -85,B 0,C 180,E1 -23151.188,E2 -23151.188} C_VEL
LIN {X 0,Y 178.641,Z 298.845,A -85,B 0,C 180,E1 -23154.995,E2 -23154.995} C_VEL
LIN {X 0,Y 179.806,Z 296.954,A -85,B 0,C 180,E1 -23156.1,E2 -23156.1} C_VEL
LIN {X 0,Y 181.062,Z 294.152,A -85,B 0,C 180,E1 -23157.698,E2 -23157.698} C_VEL
LIN {X 0,Y 181.922,Z 289.315,A -85,B 0,C 180,E1 -23160.401,E2 -23160.401} C_VEL
LIN {X 0,Y 183.067,Z 282.913,A -85,B 0,C 180,E1 -23163.527,E2 -23163.527} C_VEL
LIN {X 0,Y 183.94,Z 280.525,A -85,B 0,C 180,E1 -23164.479,E2 -23164.479} C_VEL
LIN {X 0,Y 186.745,Z 273.242,A -85,B 0,C 180,E1 -23167.024,E2 -23167.024} C_VEL
LIN {X 0,Y 188.912,Z 264.831,A -85,B 0,C 180,E1 -23169.797,E2 -23169.797} C_VEL
LIN {X 0,Y 190.199,Z 256.946,A -85,B 0,C 180,E1 -23172.351,E2 -23172.351} C_VEL
LIN {X 0,Y 190.673,Z 249.535,A -85,B 0,C 180,E1 -23174.802,E2 -23174.802} C_VEL
LIN {X 0,Y 189.967,Z 244.822,A -85,B 0,C 180,E1 -23176.81,E2 -23176.81} C_VEL
LIN {X 0,Y 188.435,Z 239.337,A -85,B 0,C 180,E1 -23179.627,E2 -23179.627} C_VEL
LIN {X 0,Y 186.286,Z 232.629,A -85,B 0,C 180,E1 -23183.747,E2 -23183.747} C_VEL
LIN {X 0,Y 184.495,Z 227.632,A -85,B 0,C 180,E1 -23187.77,E2 -23187.77} C_VEL
LIN {X 0,Y 182.909,Z 224.461,A -85,B 0,C 180,E1 -23192.098,E2 -23192.098} C_VEL
LIN {X 0,Y 182.407,Z 222.988,A -85,B 0,C 180,E1 -23194.923,E2 -23194.923} C_VEL
LIN {X 0,Y 182.243,Z 222.02,A -85,B 0,C 180,E1 -23197.751,E2 -23197.751} C_VEL
LIN {X 0,Y 182.625,Z 221.868,A -85,B 0,C 180,E1 -23202.068,E2 -23202.068} C_VEL
LIN {X 0,Y 184.212,Z 222.7,A -85,B 0,C 180,E1 -23206.766,E2 -23206.766} C_VEL
LIN {X 0,Y 186.939,Z 227.284,A -85,B 0,C 180,E1 -23212.678,E2 -23212.678} C_VEL
LIN {X 0,Y 189.445,Z 232.092,A -85,B 0,C 180,E1 -23216.809,E2 -23216.809} C_VEL
LIN {X 0,Y 191.124,Z 237.328,A -85,B 0,C 180,E1 -23219.999,E2 -23219.999} C_VEL
LIN {X 0,Y 192.252,Z 242.252,A -85,B 0,C 180,E1 -23222.618,E2 -23222.618} C_VEL
LIN {X 0,Y 192.716,Z 248.706,A -85,B 0,C 180,E1 -23225.492,E2 -23225.492} C_VEL
LIN {X 0,Y 192.404,Z 255.625,A -85,B 0,C 180,E1 -23228.4,E2 -23228.4} C_VEL
LIN {X 0,Y 192.134,Z 257.239,A -85,B 0,C 180,E1 -23229.021,E2 -23229.021} C_VEL
LIN {X 0,Y 187.826,Z 265.021,A -85,B 0,C 180,E1 -23231.318,E2 -23231.318} C_VEL
LIN {X 0,Y 183.201,Z 272.396,A -85,B 0,C 180,E1 -23234.062,E2 -23234.062} C_VEL
LIN {X 0,Y 178.186,Z 279.531,A -85,B 0,C 180,E1 -23237.531,E2 -23237.531} C_VEL
LIN {X 0,Y 173.579,Z 285.372,A -85,B 0,C 180,E1 -23241.369,E2 -23241.369} C_VEL
LIN {X 0,Y 169.351,Z 290.078,A -85,B 0,C 180,E1 -23245.948,E2 -23245.948} C_VEL
LIN {X 0,Y 166.206,Z 292.994,A -85,B 0,C 180,E1 -23250.491,E2 -23250.491} C_VEL
LIN {X 0,Y 163.838,Z 294.412,A -85,B 0,C 180,E1 -23255.409,E2 -23255.409} C_VEL
LIN {X 0,Y 162.474,Z 294.258,A -85,B 0,C 180,E1 -23260.453,E2 -23260.453} C_VEL
LIN {X 0,Y 162.041,Z 293.183,A -85,B 0,C 180,E1 -23263.941,E2 -23263.941} C_VEL
LIN {X 0,Y 162.01,Z 291.27,A -85,B 0,C 180,E1 -23267.513,E2 -23267.513} C_VEL
LIN {X 0,Y 162.475,Z 288.445,A -85,B 0,C 180,E1 -23271.131,E2 -23271.131} C_VEL
LIN {X 0,Y 163.363,Z 284.547,A -85,B 0,C 180,E1 -23274.823,E2 -23274.823} C_VEL
LIN {X 0,Y 164.871,Z 278.366,A -85,B 0,C 180,E1 -23279.234,E2 -23279.234} C_VEL
LIN {X 0,Y 166.794,Z 271.044,A -85,B 0,C 180,E1 -23283.181,E2 -23283.181} C_VEL
LIN {X 0,Y 169.259,Z 262.404,A -85,B 0,C 180,E1 -23286.821,E2 -23286.821} C_VEL
LIN {X 0,Y 171.944,Z 252.558,A -85,B 0,C 180,E1 -23290.063,E2 -23290.063} C_VEL
LIN {X 0,Y 174.443,Z 242.435,A -85,B 0,C 180,E1 -23292.714,E2 -23292.714} C_VEL
LIN {X 0,Y 175.82,Z 235.561,A -85,B 0,C 180,E1 -23294.233,E2 -23294.233} C_VEL
LIN {X 0,Y 174.025,Z 224.029,A -85,B 0,C 180,E1 -23296.869,E2 -23296.869} C_VEL
LIN {X 0,Y 171.824,Z 213.406,A -85,B 0,C 180,E1 -23299.001,E2 -23299.001} C_VEL
LIN {X 0,Y 169.179,Z 203.97,A -85,B 0,C 180,E1 -23300.736,E2 -23300.736} C_VEL
LIN {X 0,Y 165.552,Z 194.546,A -85,B 0,C 180,E1 -23302.414,E2 -23302.414} C_VEL
LIN {X 0,Y 164.741,Z 191.967,A -85,B 0,C 180,E1 -23302.877,E2 -23302.877} C_VEL
LIN {X 0,Y 165.041,Z 191.925,A -85,B 0,C 180,E1 -23307.559,E2 -23307.559} C_VEL
LIN {X 0,Y 165.294,Z 191.893,A -85,B 0,C 180,E1 -23310,E2 -23310} C_VEL
LIN {X 0,Y 164.773,Z 191.955,A -85,B 0,C 180,E1 -23314.893,E2 -23314.893} C_VEL
LIN {X 0,Y 164.859,Z 191.952,A -85,B 0,C 180,E1 -23317.347,E2 -23317.347} C_VEL
LIN {X 0,Y 164.777,Z 191.956,A -85,B 0,C 180,E1 -23321.198,E2 -23321.198} C_VEL
LIN {X 0,Y 164.523,Z 191.989,A -85,B 0,C 180,E1 -23327.398,E2 -23327.398} C_VEL
LIN {X 0,Y 164.517,Z 191.996,A -85,B 0,C 180,E1 -23329.983,E2 -23329.983} C_VEL
LIN {X 0,Y 164.39,Z 191.998,A -85,B 0,C 180,E1 -23336.134,E2 -23336.134} C_VEL
LIN {X 0,Y 164.371,Z 192.013,A -85,B 0,C 180,E1 -23341.227,E2 -23341.227} C_VEL
LIN {X 0,Y 164.291,Z 192.006,A -85,B 0,C 180,E1 -23346.79,E2 -23346.79} C_VEL
LIN {X 0,Y 164.288,Z 192.018,A -85,B 0,C 180,E1 -23349.917,E2 -23349.917} C_VEL
LIN {X 0,Y 164.276,Z 192.021,A -85,B 0,C 180,E1 -23353.343,E2 -23353.343} C_VEL
LIN {X 0,Y 164.29,Z 192.007,A -85,B 0,C 180,E1 -23356.809,E2 -23356.809} C_VEL
LIN {X 0,Y 164.293,Z 192.01,A -85,B 0,C 180,E1 -23360.353,E2 -23360.353} C_VEL
LIN {X 0,Y 164.328,Z 192.015,A -85,B 0,C 180,E1 -23364.35,E2 -23364.35} C_VEL
LIN {X 0,Y 164.387,Z 191.996,A -85,B 0,C 180,E1 -23369.135,E2 -23369.135} C_VEL
LIN {X 0,Y 164.417,Z 191.998,A -85,B 0,C 180,E1 -23374.696,E2 -23374.696} C_VEL
LIN {X 0,Y 164.519,Z 191.989,A -85,B 0,C 180,E1 -23380.018,E2 -23380.018} C_VEL
LIN {X 0,Y 164.53,Z 191.973,A -85,B 0,C 180,E1 -23385.151,E2 -23385.151} C_VEL
LIN {X 0,Y 164.768,Z 191.96,A -85,B 0,C 180,E1 -23390.178,E2 -23390.178} C_VEL
LIN {X 0,Y 164.832,Z 191.951,A -85,B 0,C 180,E1 -23392.652,E2 -23392.652} C_VEL
LIN {X 0,Y 165.049,Z 191.908,A -85,B 0,C 180,E1 -23397.561,E2 -23397.561} C_VEL
LIN {X 0,Y 165.296,Z 191.887,A -85,B 0,C 180,E1 -23400.001,E2 -23400.001} C_VEL
LIN {X 0,Y 164.76,Z 191.96,A -85,B 0,C 180,E1 -23404.895,E2 -23404.895} C_VEL
LIN {X 0,Y 164.828,Z 191.945,A -85,B 0,C 180,E1 -23407.35,E2 -23407.35} C_VEL
LIN {X 0,Y 164.619,Z 191.979,A -85,B 0,C 180,E1 -23412.327,E2 -23412.327} C_VEL
LIN {X 0,Y 164.526,Z 191.983,A -85,B 0,C 180,E1 -23417.4,E2 -23417.4} C_VEL
LIN {X 0,Y 164.522,Z 191.989,A -85,B 0,C 180,E1 -23419.984,E2 -23419.984} C_VEL
LIN {X 0,Y 164.395,Z 192.008,A -85,B 0,C 180,E1 -23426.135,E2 -23426.135} C_VEL
LIN {X 0,Y 164.435,Z 192.046,A -85,B 0,C 180,E1 -23431.262,E2 -23431.262} C_VEL
LIN {X 0,Y 165.002,Z 195.582,A -85,B 0,C 180,E1 -23436.607,E2 -23436.607} C_VEL
LIN {X 0,Y 165.455,Z 198.043,A -85,B 0,C 180,E1 -23440.131,E2 -23440.131} C_VEL
LIN {X 0,Y 166.017,Z 200.828,A -85,B 0,C 180,E1 -23443.974,E2 -23443.974} C_VEL
LIN {X 0,Y 166.601,Z 203.566,A -85,B 0,C 180,E1 -23447.55,E2 -23447.55} C_VEL
LIN {X 0,Y 166.978,Z 206.996,A -85,B 0,C 180,E1 -23451.803,E2 -23451.803} C_VEL
LIN {X 0,Y 169.268,Z 219.221,A -85,B 0,C 180,E1 -23453.318,E2 -23453.318} C_VEL
LIN {X 0,Y 170.96,Z 232.695,A -85,B 0,C 180,E1 -23455.306,E2 -23455.306} C_VEL
LIN {X 0,Y 171.841,Z 245.571,A -85,B 0,C 180,E1 -23457.614,E2 -23457.614} C_VEL
LIN {X 0,Y 172.156,Z 255.62,A -85,B 0,C 180,E1 -23459.778,E2 -23459.778} C_VEL
LIN {X 0,Y 172.085,Z 265.694,A -85,B 0,C 180,E1 -23462.319,E2 -23462.319} C_VEL
LIN {X 0,Y 171.62,Z 270.111,A -85,B 0,C 180,E1 -23463.555,E2 -23463.555} C_VEL
LIN {X 0,Y 169.123,Z 278.923,A -85,B 0,C 180,E1 -23466.3,E2 -23466.3} C_VEL
LIN {X 0,Y 166.76,Z 287.472,A -85,B 0,C 180,E1 -23469.654,E2 -23469.654} C_VEL
LIN {X 0,Y 164.732,Z 294.759,A -85,B 0,C 180,E1 -23473.264,E2 -23473.264} C_VEL
LIN {X 0,Y 163.183,Z 301.441,A -85,B 0,C 180,E1 -23477.565,E2 -23477.565} C_VEL
LIN {X 0,Y 162.487,Z 305.826,A -85,B 0,C 180,E1 -23481.293,E2 -23481.293} C_VEL
LIN {X 0,Y 162.297,Z 309.107,A -85,B 0,C 180,E1 -23485.032,E2 -23485.032} C_VEL
LIN {X 0,Y 162.323,Z 310.702,A -85,B 0,C 180,E1 -23487.519,E2 -23487.519} C_VEL
LIN {X 0,Y 162.351,Z 311.866,A -85,B 0,C 180,E1 -23490,E2 -23490} C_VEL
LIN {X 0,Y 162.112,Z 312.865,A -85,B 0,C 180,E1 -23494.34,E2 -23494.34} C_VEL
LIN {X 0,Y 162.15,Z 312.819,A -85,B 0,C 180,E1 -23497.472,E2 -23497.472} C_VEL
LIN {X 0,Y 163.078,Z 311.545,A -85,B 0,C 180,E1 -23502.444,E2 -23502.444} C_VEL
LIN {X 0,Y 163.883,Z 310.347,A -85,B 0,C 180,E1 -23504.911,E2 -23504.911} C_VEL
LIN {X 0,Y 166.627,Z 306.736,A -85,B 0,C 180,E1 -23509.721,E2 -23509.721} C_VEL
LIN {X 0,Y 169.401,Z 302.972,A -85,B 0,C 180,E1 -23513.212,E2 -23513.212} C_VEL
LIN {X 0,Y 173.272,Z 297.534,A -85,B 0,C 180,E1 -23516.969,E2 -23516.969} C_VEL
LIN {X 0,Y 177.498,Z 291.169,A -85,B 0,C 180,E1 -23520.321,E2 -23520.321} C_VEL
LIN {X 0,Y 182.333,Z 283.708,A -85,B 0,C 180,E1 -23523.317,E2 -23523.317} C_VEL
LIN {X 0,Y 183.94,Z 280.525,A -85,B 0,C 180,E1 -23524.479,E2 -23524.479} C_VEL
LIN {X 0,Y 184.888,Z 277.015,A -85,B 0,C 180,E1 -23525.922,E2 -23525.922} C_VEL
LIN {X 0,Y 184.91,Z 273.733,A -85,B 0,C 180,E1 -23527.459,E2 -23527.459} C_VEL
LIN {X 0,Y 184.068,Z 264.926,A -85,B 0,C 180,E1 -23531.625,E2 -23531.625} C_VEL
LIN {X 0,Y 184.392,Z 262.401,A -85,B 0,C 180,E1 -23532.591,E2 -23532.591} C_VEL
LIN {X 0,Y 185.567,Z 254.463,A -85,B 0,C 180,E1 -23535.352,E2 -23535.352} C_VEL
LIN {X 0,Y 185.465,Z 250.616,A -85,B 0,C 180,E1 -23536.991,E2 -23536.991} C_VEL
LIN {X 0,Y 184.14,Z 244.621,A -85,B 0,C 180,E1 -23540.254,E2 -23540.254} C_VEL
LIN {X 0,Y 182.327,Z 237.986,A -85,B 0,C 180,E1 -23544.675,E2 -23544.675} C_VEL
LIN {X 0,Y 180.983,Z 233.361,A -85,B 0,C 180,E1 -23548.685,E2 -23548.685} C_VEL
LIN {X 0,Y 179.951,Z 231.014,A -85,B 0,C 180,E1 -23552.051,E2 -23552.051} C_VEL
LIN {X 0,Y 179.354,Z 228.779,A -85,B 0,C 180,E1 -23556.929,E2 -23556.929} C_VEL
LIN {X 0,Y 179.473,Z 228.293,A -85,B 0,C 180,E1 -23560.023,E2 -23560.023} C_VEL
LIN {X 0,Y 181.087,Z 229.066,A -85,B 0,C 180,E1 -23566.533,E2 -23566.533} C_VEL
LIN {X 0,Y 182.738,Z 232.278,A -85,B 0,C 180,E1 -23571.149,E2 -23571.149} C_VEL
LIN {X 0,Y 184.934,Z 236.771,A -85,B 0,C 180,E1 -23575.64,E2 -23575.64} C_VEL
LIN {X 0,Y 185.857,Z 239.814,A -85,B 0,C 180,E1 -23577.832,E2 -23577.832} C_VEL
LIN {X 0,Y 187.045,Z 245.14,A -85,B 0,C 180,E1 -23581.075,E2 -23581.075} C_VEL
LIN {X 0,Y 187.342,Z 249.921,A -85,B 0,C 180,E1 -23583.494,E2 -23583.494} C_VEL
LIN {X 0,Y 187.032,Z 256.317,A -85,B 0,C 180,E1 -23586.472,E2 -23586.472} C_VEL
LIN {X 0,Y 186.698,Z 258.693,A -85,B 0,C 180,E1 -23587.532,E2 -23587.532} C_VEL
LIN {X 0,Y 186.039,Z 260.26,A -85,B 0,C 180,E1 -23588.087,E2 -23588.087} C_VEL
LIN {X 0,Y 181.211,Z 268.157,A -85,B 0,C 180,E1 -23590.615,E2 -23590.615} C_VEL
LIN {X 0,Y 175.753,Z 276.018,A -85,B 0,C 180,E1 -23593.881,E2 -23593.881} C_VEL
LIN {X 0,Y 170.881,Z 282.192,A -85,B 0,C 180,E1 -23597.331,E2 -23597.331} C_VEL
LIN {X 0,Y 166.096,Z 287.56,A -85,B 0,C 180,E1 -23601.426,E2 -23601.426} C_VEL
LIN {X 0,Y 162.287,Z 291.332,A -85,B 0,C 180,E1 -23605.66,E2 -23605.66} C_VEL
LIN {X 0,Y 159.977,Z 293.238,A -85,B 0,C 180,E1 -23608.896,E2 -23608.896} C_VEL
LIN {X 0,Y 158.029,Z 294.471,A -85,B 0,C 180,E1 -23612.329,E2 -23612.329} C_VEL
LIN {X 0,Y 156.484,Z 294.997,A -85,B 0,C 180,E1 -23616.058,E2 -23616.058} C_VEL
LIN {X 0,Y 155.5,Z 294.71,A -85,B 0,C 180,E1 -23619.794,E2 -23619.794} C_VEL
LIN {X 0,Y 154.986,Z 293.609,A -85,B 0,C 180,E1 -23623.486,E2 -23623.486} C_VEL
LIN {X 0,Y 154.922,Z 291.737,A -85,B 0,C 180,E1 -23627.119,E2 -23627.119} C_VEL
LIN {X 0,Y 155.29,Z 289.12,A -85,B 0,C 180,E1 -23630.683,E2 -23630.683} C_VEL
LIN {X 0,Y 156.045,Z 285.751,A -85,B 0,C 180,E1 -23634.161,E2 -23634.161} C_VEL
LIN {X 0,Y 157.243,Z 280.755,A -85,B 0,C 180,E1 -23638.123,E2 -23638.123} C_VEL
LIN {X 0,Y 159.003,Z 274.232,A -85,B 0,C 180,E1 -23642.127,E2 -23642.127} C_VEL
LIN {X 0,Y 161.431,Z 265.948,A -85,B 0,C 180,E1 -23646.096,E2 -23646.096} C_VEL
LIN {X 0,Y 164.189,Z 256.364,A -85,B 0,C 180,E1 -23649.648,E2 -23649.648} C_VEL
LIN {X 0,Y 166.812,Z 246.576,A -85,B 0,C 180,E1 -23652.531,E2 -23652.531} C_VEL
LIN {X 0,Y 169.044,Z 237.073,A -85,B 0,C 180,E1 -23654.792,E2 -23654.792} C_VEL
LIN {X 0,Y 167.389,Z 225.612,A -85,B 0,C 180,E1 -23657.574,E2 -23657.574} C_VEL
LIN {X 0,Y 165.232,Z 214.723,A -85,B 0,C 180,E1 -23659.898,E2 -23659.898} C_VEL
LIN {X 0,Y 162.334,Z 204.797,A -85,B 0,C 180,E1 -23661.848,E2 -23661.848} C_VEL
LIN {X 0,Y 158.702,Z 195.683,A -85,B 0,C 180,E1 -23663.603,E2 -23663.603} C_VEL
LIN {X 0,Y 157.682,Z 192.845,A -85,B 0,C 180,E1 -23664.164,E2 -23664.164} C_VEL
LIN {X 0,Y 158.256,Z 192.77,A -85,B 0,C 180,E1 -23670,E2 -23670} C_VEL
LIN {X 0,Y 157.822,Z 192.83,A -85,B 0,C 180,E1 -23677.677,E2 -23677.677} C_VEL
LIN {X 0,Y 157.703,Z 192.838,A -85,B 0,C 180,E1 -23681.362,E2 -23681.362} C_VEL
LIN {X 0,Y 157.485,Z 192.872,A -85,B 0,C 180,E1 -23685.531,E2 -23685.531} C_VEL
LIN {X 0,Y 157.413,Z 192.881,A -85,B 0,C 180,E1 -23690.926,E2 -23690.926} C_VEL
LIN {X 0,Y 157.311,Z 192.879,A -85,B 0,C 180,E1 -23696.685,E2 -23696.685} C_VEL
LIN {X 0,Y 157.271,Z 192.895,A -85,B 0,C 180,E1 -23702.428,E2 -23702.428} C_VEL
LIN {X 0,Y 157.265,Z 192.881,A -85,B 0,C 180,E1 -23706.45,E2 -23706.45} C_VEL
LIN {X 0,Y 157.208,Z 192.902,A -85,B 0,C 180,E1 -23712.111,E2 -23712.111} C_VEL
LIN {X 0,Y 157.208,Z 192.884,A -85,B 0,C 180,E1 -23717.89,E2 -23717.89} C_VEL
LIN {X 0,Y 157.265,Z 192.894,A -85,B 0,C 180,E1 -23723.552,E2 -23723.552} C_VEL
LIN {X 0,Y 157.29,Z 192.886,A -85,B 0,C 180,E1 -23728.097,E2 -23728.097} C_VEL
LIN {X 0,Y 157.32,Z 192.879,A -85,B 0,C 180,E1 -23733.467,E2 -23733.467} C_VEL
LIN {X 0,Y 157.446,Z 192.87,A -85,B 0,C 180,E1 -23739.617,E2 -23739.617} C_VEL
